LIN {X -0.130,Y -407.420,Z 765.576,A 0.000,B 0.000,C 90.000,E1 139.666} C_DIS
LIN {X -0.060,Y -413.085,Z 765.572,A 0.000,B 0.000,C 90.000,E1 138.976} C_DIS
LIN {X 0.241,Y -427.502,Z 765.564,A 0.000,B 0.000,C 90.000,E1 137.391} C_DIS
LIN {X 0.053,Y -436.215,Z 765.559,A 0.000,B 0.000,C 90.000,E1 136.539} C_DIS
LIN {X 0.009,Y -443.347,Z 765.555,A 0.000,B 0.000,C 90.000,E1 135.810} C_DIS
LIN {X -0.045,Y -451.801,Z 765.550,A 0.000,B 0.000,C 90.000,E1 134.919} C_DIS
LIN {X 0.010,Y -457.316,Z 765.546,A 0.000,B 0.000,C 90.000,E1 134.312} C_DIS
LIN {X 0.124,Y -465.443,Z 765.541,A 0.000,B 0.000,C 90.000,E1 133.380} C_DIS
LIN {X 0.124,Y -473.358,Z 765.536,A 0.000,B 0.000,C 90.000,E1 132.447} C_DIS
LIN {X -0.077,Y -480.793,Z 765.531,A 0.000,B 0.000,C 90.000,E1 131.553} C_DIS
LIN {X -0.084,Y -486.838,Z 765.527,A 0.000,B 0.000,C 90.000,E1 130.782} C_DIS
LIN {X 0.149,Y -492.370,Z 765.522,A 0.000,B 0.000,C 90.000,E1 130.011} C_DIS
LIN {X 0.158,Y -496.618,Z 765.519,A 0.000,B 0.000,C 90.000,E1 129.402} C_DIS
LIN {X 0.003,Y -502.509,Z 765.514,A 0.000,B 0.000,C 90.000,E1 128.543} C_DIS
LIN {X -0.097,Y -507.241,Z 765.510,A 0.000,B 0.000,C 90.000,E1 127.810} C_DIS
LIN {X -0.187,Y -511.626,Z 765.506,A 0.000,B 0.000,C 90.000,E1 127.076} C_DIS
LIN {X 0.175,Y -515.816,Z 765.502,A 0.000,B 0.000,C 90.000,E1 126.297} C_DIS
LIN {X -0.201,Y -521.468,Z 765.496,A 0.000,B 0.000,C 90.000,E1 125.311} C_DIS
LIN {X 0.259,Y -525.137,Z 765.492,A 0.000,B 0.000,C 90.000,E1 124.532} C_DIS
LIN {X -0.142,Y -529.163,Z 765.487,A 0.000,B 0.000,C 90.000,E1 123.706} C_DIS
LIN {X -0.224,Y -534.731,Z 765.480,A 0.000,B 0.000,C 90.000,E1 122.418} C_DIS
LIN {X -0.076,Y -538.231,Z 765.475,A 0.000,B 0.000,C 90.000,E1 121.544} C_DIS
LIN {X 0.107,Y -541.496,Z 765.471,A 0.000,B 0.000,C 90.000,E1 120.669} C_DIS
LIN {X 0.325,Y -544.507,Z 765.466,A 0.000,B 0.000,C 90.000,E1 119.795} C_DIS
LIN {X -0.175,Y -547.339,Z 765.461,A 0.000,B 0.000,C 90.000,E1 118.999} C_DIS
LIN {X 0.079,Y -550.940,Z 765.455,A 0.000,B 0.000,C 90.000,E1 117.847} C_DIS
LIN {X -0.134,Y -552.669,Z 765.452,A 0.000,B 0.000,C 90.000,E1 117.308} C_DIS
LIN {X 0.175,Y -554.965,Z 765.447,A 0.000,B 0.000,C 90.000,E1 116.437} C_DIS
LIN {X 0.048,Y -557.323,Z 765.441,A 0.000,B 0.000,C 90.000,E1 115.335} C_DIS
LIN {X 0.126,Y -558.444,Z 765.438,A 0.000,B 0.000,C 90.000,E1 114.771} C_DIS
LIN {X -0.202,Y -560.084,Z 765.432,A 0.000,B 0.000,C 90.000,E1 113.695} C_DIS
LIN {X 0.098,Y -561.976,Z 765.424,A 0.000,B 0.000,C 90.000,E1 112.280} C_DIS
LIN {X 0.121,Y -563.367,Z 765.418,A 0.000,B 0.000,C 90.000,E1 111.173} C_DIS
LIN {X -0.041,Y -564.984,Z 765.410,A 0.000,B 0.000,C 90.000,E1 109.812} C_DIS
LIN {X -0.175,Y -566.142,Z 765.404,A 0.000,B 0.000,C 90.000,E1 108.725} C_DIS
LIN {X 0.038,Y -567.477,Z 765.396,A 0.000,B 0.000,C 90.000,E1 107.330} C_DIS
LIN {X 0.267,Y -568.968,Z 765.387,A 0.000,B 0.000,C 90.000,E1 105.662} C_DIS
LIN {X -0.165,Y -570.428,Z 765.378,A 0.000,B 0.000,C 90.000,E1 104.064} C_DIS
LIN {X -0.194,Y -572.542,Z 765.366,A 0.000,B 0.000,C 90.000,E1 101.883} C_DIS
LIN {X -0.244,Y -574.082,Z 765.357,A 0.000,B 0.000,C 90.000,E1 100.254} C_DIS
LIN {X -0.098,Y -575.102,Z 765.351,A 0.000,B 0.000,C 90.000,E1 99.151} C_DIS
LIN {X 0.269,Y -576.268,Z 765.343,A 0.000,B 0.000,C 90.000,E1 97.757} C_DIS
LIN {X -0.234,Y -577.702,Z 765.333,A 0.000,B 0.000,C 90.000,E1 95.910} C_DIS
LIN {X 0.187,Y -578.800,Z 765.324,A 0.000,B 0.000,C 90.000,E1 94.245} C_DIS
LIN {X -0.104,Y -579.695,Z 765.316,A 0.000,B 0.000,C 90.000,E1 92.922} C_DIS
LIN {X -0.251,Y -580.601,Z 765.307,A 0.000,B 0.000,C 90.000,E1 91.318} C_DIS
LIN {X 0.192,Y -581.406,Z 765.298,A 0.000,B 0.000,C 90.000,E1 89.656} C_DIS
LIN {X 0.084,Y -582.021,Z 765.289,A 0.000,B 0.000,C 90.000,E1 88.051} C_DIS
LIN {X -0.182,Y -582.433,Z 765.282,A 0.000,B 0.000,C 90.000,E1 86.731} C_DIS
LIN {X -0.066,Y -582.897,Z 765.271,A 0.000,B 0.000,C 90.000,E1 84.837} C_DIS
LIN {X -0.290,Y -583.123,Z 765.264,A 0.000,B 0.000,C 90.000,E1 83.514} C_DIS
LIN {X 0.019,Y -583.259,Z 765.253,A 0.000,B 0.000,C 90.000,E1 81.602} C_DIS
LIN {X 0.060,Y -583.261,Z 765.249,A 0.000,B 0.000,C 90.000,E1 80.792} C_DIS
LIN {X -0.001,Y -583.262,Z 765.241,A 0.000,B 0.000,C 90.000,E1 79.454} C_DIS
LIN {X -0.070,Y -583.092,Z 765.234,A 0.000,B 0.000,C 90.000,E1 78.117} C_DIS
LIN {X 0.003,Y -582.582,Z 765.224,A 0.000,B 0.000,C 90.000,E1 76.228} C_DIS
LIN {X 0.178,Y -582.150,Z 765.216,A 0.000,B 0.000,C 90.000,E1 74.866} C_DIS
LIN {X -0.220,Y -581.615,Z 765.209,A 0.000,B 0.000,C 90.000,E1 73.559} C_DIS
LIN {X -0.251,Y -580.809,Z 765.200,A 0.000,B 0.000,C 90.000,E1 71.945} C_DIS
LIN {X 0.223,Y -580.086,Z 765.192,A 0.000,B 0.000,C 90.000,E1 70.550} C_DIS
LIN {X -0.250,Y -579.363,Z 765.186,A 0.000,B 0.000,C 90.000,E1 69.518} C_DIS
LIN {X -0.141,Y -578.400,Z 765.179,A 0.000,B 0.000,C 90.000,E1 68.156} C_DIS
LIN {X -0.044,Y -577.275,Z 765.171,A 0.000,B 0.000,C 90.000,E1 66.794} C_DIS
LIN {X 0.035,Y -576.497,Z 765.167,A 0.000,B 0.000,C 90.000,E1 65.973} C_DIS
LIN {X -0.286,Y -575.321,Z 765.161,A 0.000,B 0.000,C 90.000,E1 64.921} C_DIS
LIN {X -0.133,Y -574.053,Z 765.155,A 0.000,B 0.000,C 90.000,E1 63.819} C_DIS
LIN {X -0.090,Y -572.965,Z 765.150,A 0.000,B 0.000,C 90.000,E1 62.999} C_DIS
LIN {X 0.035,Y -571.306,Z 765.144,A 0.000,B 0.000,C 90.000,E1 61.897} C_DIS
LIN {X 0.135,Y -569.356,Z 765.138,A 0.000,B 0.000,C 90.000,E1 60.795} C_DIS
LIN {X -0.293,Y -567.145,Z 765.132,A 0.000,B 0.000,C 90.000,E1 59.744} C_DIS
LIN {X 0.111,Y -565.957,Z 765.129,A 0.000,B 0.000,C 90.000,E1 59.154} C_DIS
LIN {X -0.078,Y -563.214,Z 765.123,A 0.000,B 0.000,C 90.000,E1 58.074} C_DIS
LIN {X 0.002,Y -560.097,Z 765.117,A 0.000,B 0.000,C 90.000,E1 56.962} C_DIS
LIN {X -0.039,Y -557.565,Z 765.112,A 0.000,B 0.000,C 90.000,E1 56.135} C_DIS
LIN {X -0.185,Y -555.830,Z 765.109,A 0.000,B 0.000,C 90.000,E1 55.595} C_DIS
LIN {X -0.274,Y -552.875,Z 765.104,A 0.000,B 0.000,C 90.000,E1 54.769} C_DIS
LIN {X -0.076,Y -549.494,Z 765.099,A 0.000,B 0.000,C 90.000,E1 53.909} C_DIS
LIN {X -0.102,Y -546.409,Z 765.096,A 0.000,B 0.000,C 90.000,E1 53.210} C_DIS
LIN {X 0.168,Y -543.046,Z 765.092,A 0.000,B 0.000,C 90.000,E1 52.477} C_DIS
LIN {X 0.228,Y -540.213,Z 765.089,A 0.000,B 0.000,C 90.000,E1 51.904} C_DIS
LIN {X -0.155,Y -537.096,Z 765.085,A 0.000,B 0.000,C 90.000,E1 51.376} C_DIS
LIN {X 0.028,Y -532.761,Z 765.081,A 0.000,B 0.000,C 90.000,E1 50.642} C_DIS
LIN {X 0.008,Y -528.850,Z 765.078,A 0.000,B 0.000,C 90.000,E1 50.070} C_DIS
LIN {X -0.118,Y -524.929,Z 765.075,A 0.000,B 0.000,C 90.000,E1 49.542} C_DIS
LIN {X 0.141,Y -520.019,Z 765.072,A 0.000,B 0.000,C 90.000,E1 48.933} C_DIS
LIN {X -0.100,Y -516.148,Z 765.070,A 0.000,B 0.000,C 90.000,E1 48.528} C_DIS
LIN {X -0.016,Y -510.601,Z 765.066,A 0.000,B 0.000,C 90.000,E1 47.957} C_DIS
LIN {X -0.040,Y -506.284,Z 765.064,A 0.000,B 0.000,C 90.000,E1 47.553} C_DIS
LIN {X 0.083,Y -500.284,Z 765.061,A 0.000,B 0.000,C 90.000,E1 47.025} C_DIS
LIN {X 0.034,Y -495.791,Z 765.059,A 0.000,B 0.000,C 90.000,E1 46.662} C_DIS
LIN {X 0.187,Y -487.760,Z 765.056,A 0.000,B 0.000,C 90.000,E1 46.053} C_DIS
LIN {X -0.185,Y -481.381,Z 765.054,A 0.000,B 0.000,C 90.000,E1 45.648} C_DIS
LIN {X 0.041,Y -473.279,Z 765.051,A 0.000,B 0.000,C 90.000,E1 45.081} C_DIS
LIN {X 0.063,Y -463.499,Z 765.047,A 0.000,B 0.000,C 90.000,E1 44.433} C_DIS
LIN {X 0.134,Y -444.156,Z 765.040,A 0.000,B 0.000,C 90.000,E1 43.137} C_DIS
LIN {X -0.050,Y -419.026,Z 765.030,A 0.000,B 0.000,C 90.000,E1 41.353} C_DIS
LIN {X 0.070,Y -413.289,Z 765.027,A 0.000,B 0.000,C 90.000,E1 40.862} C_DIS
LIN {X -0.212,Y -409.341,Z 765.025,A 0.000,B 0.000,C 90.000,E1 40.539} C_DIS
LIN {X -0.238,Y -409.310,Z 765.025,A 0.000,B 0.000,C 90.000,E1 40.539} C_DIS
LIN {X 0.130,Y -406.118,Z 765.015,A 0.000,B 0.000,C 90.000,E1 38.624} C_DIS
LIN {X 0.096,Y -404.664,Z 765.011,A 0.000,B 0.000,C 90.000,E1 37.935} C_DIS
LIN {X 0.157,Y -399.374,Z 764.996,A 0.000,B 0.000,C 90.000,E1 35.311} C_DIS
LIN {X 0.042,Y -399.270,Z 764.994,A 0.000,B 0.000,C 90.000,E1 34.978} C_DIS
LIN {X -0.237,Y -399.849,Z 764.979,A 0.000,B 0.000,C 90.000,E1 32.212} C_DIS
LIN {X -0.249,Y -400.946,Z 764.963,A 0.000,B 0.000,C 90.000,E1 29.411} C_DIS
LIN {X 0.141,Y -402.082,Z 764.952,A 0.000,B 0.000,C 90.000,E1 27.257} C_DIS
LIN {X 0.160,Y -403.832,Z 764.936,A 0.000,B 0.000,C 90.000,E1 24.463} C_DIS
LIN {X -0.098,Y -405.866,Z 764.921,A 0.000,B 0.000,C 90.000,E1 21.716} C_DIS
LIN {X -0.097,Y -409.099,Z 764.903,A 0.000,B 0.000,C 90.000,E1 18.598} C_DIS
LIN {X -0.112,Y -412.740,Z 764.888,A 0.000,B 0.000,C 90.000,E1 15.843} C_DIS
LIN {X 0.131,Y -416.278,Z 764.875,A 0.000,B 0.000,C 90.000,E1 13.411} C_DIS
LIN {X -0.213,Y -420.108,Z 764.861,A 0.000,B 0.000,C 90.000,E1 11.074} C_DIS
LIN {X 0.219,Y -422.884,Z 764.852,A 0.000,B 0.000,C 90.000,E1 9.321} C_DIS
LIN {X 0.150,Y -425.769,Z 764.843,A 0.000,B 0.000,C 90.000,E1 7.644} C_DIS
LIN {X 0.190,Y -429.171,Z 764.831,A 0.000,B 0.000,C 90.000,E1 5.625} C_DIS
LIN {X -0.163,Y -432.714,Z 764.820,A 0.000,B 0.000,C 90.000,E1 3.669} C_DIS
LIN {X -0.145,Y -435.835,Z 764.811,A 0.000,B 0.000,C 90.000,E1 2.007} C_DIS
LIN {X -0.158,Y -440.762,Z 764.797,A 0.000,B 0.000,C 90.000,E1 359.484} C_DIS
LIN {X -0.165,Y -445.509,Z 764.784,A 0.000,B 0.000,C 90.000,E1 357.192} C_DIS
LIN {X 0.010,Y -450.602,Z 764.772,A 0.000,B 0.000,C 90.000,E1 354.894} C_DIS
LIN {X 0.002,Y -454.397,Z 764.763,A 0.000,B 0.000,C 90.000,E1 353.280} C_DIS
LIN {X -0.098,Y -457.326,Z 764.756,A 0.000,B 0.000,C 90.000,E1 352.008} C_DIS
LIN {X 0.064,Y -459.484,Z 764.750,A 0.000,B 0.000,C 90.000,E1 351.027} C_DIS
LIN {X 0.111,Y -462.231,Z 764.743,A 0.000,B 0.000,C 90.000,E1 349.746} C_DIS
LIN {X 0.002,Y -465.459,Z 764.734,A 0.000,B 0.000,C 90.000,E1 348.173} C_DIS
LIN {X 0.238,Y -470.085,Z 764.722,A 0.000,B 0.000,C 90.000,E1 345.936} C_DIS
LIN {X -0.012,Y -471.853,Z 764.719,A 0.000,B 0.000,C 90.000,E1 345.338} C_DIS
LIN {X 0.085,Y -474.238,Z 764.715,A 0.000,B 0.000,C 90.000,E1 344.700} C_DIS
LIN {X 0.057,Y -476.137,Z 764.713,A 0.000,B 0.000,C 90.000,E1 344.338} C_DIS
LIN {X 0.276,Y -479.563,Z 764.710,A 0.000,B 0.000,C 90.000,E1 343.795} C_DIS
LIN {X 0.118,Y -482.087,Z 764.708,A 0.000,B 0.000,C 90.000,E1 343.504} C_DIS
LIN {X 0.132,Y -488.837,Z 764.705,A 0.000,B 0.000,C 90.000,E1 342.851} C_DIS
LIN {X 0.042,Y -500.528,Z 764.700,A 0.000,B 0.000,C 90.000,E1 342.000} C_DIS
LIN {X 0.262,Y -520.919,Z 764.692,A 0.000,B 0.000,C 90.000,E1 340.604} C_DIS
LIN {X 0.061,Y -536.973,Z 764.687,A 0.000,B 0.000,C 90.000,E1 339.645} C_DIS
LIN {X -0.064,Y -544.553,Z 764.684,A 0.000,B 0.000,C 90.000,E1 339.156} C_DIS
LIN {X 0.005,Y -549.016,Z 764.682,A 0.000,B 0.000,C 90.000,E1 338.827} C_DIS
LIN {X 0.092,Y -554.622,Z 764.680,A 0.000,B 0.000,C 90.000,E1 338.358} C_DIS
LIN {X 0.279,Y -560.032,Z 764.677,A 0.000,B 0.000,C 90.000,E1 337.847} C_DIS
LIN {X -0.005,Y -566.398,Z 764.674,A 0.000,B 0.000,C 90.000,E1 337.230} C_DIS
LIN {X -0.127,Y -571.260,Z 764.671,A 0.000,B 0.000,C 90.000,E1 336.719} C_DIS
LIN {X -0.173,Y -575.976,Z 764.668,A 0.000,B 0.000,C 90.000,E1 336.177} C_DIS
LIN {X 0.121,Y -579.324,Z 764.665,A 0.000,B 0.000,C 90.000,E1 335.741} C_DIS
LIN {X 0.169,Y -586.780,Z 764.660,A 0.000,B 0.000,C 90.000,E1 334.793} C_DIS
LIN {X -0.119,Y -591.775,Z 764.656,A 0.000,B 0.000,C 90.000,E1 334.152} C_DIS
LIN {X 0.077,Y -598.389,Z 764.651,A 0.000,B 0.000,C 90.000,E1 333.204} C_DIS
LIN {X 0.096,Y -604.793,Z 764.646,A 0.000,B 0.000,C 90.000,E1 332.281} C_DIS
LIN {X -0.092,Y -610.829,Z 764.641,A 0.000,B 0.000,C 90.000,E1 331.385} C_DIS
LIN {X 0.059,Y -618.094,Z 764.635,A 0.000,B 0.000,C 90.000,E1 330.205} C_DIS
LIN {X 0.329,Y -622.066,Z 764.631,A 0.000,B 0.000,C 90.000,E1 329.537} C_DIS
LIN {X 0.106,Y -627.280,Z 764.626,A 0.000,B 0.000,C 90.000,E1 328.663} C_DIS
LIN {X -0.058,Y -632.249,Z 764.621,A 0.000,B 0.000,C 90.000,E1 327.788} C_DIS
LIN {X -0.184,Y -636.241,Z 764.617,A 0.000,B 0.000,C 90.000,E1 327.041} C_DIS
LIN {X 0.120,Y -641.152,Z 764.611,A 0.000,B 0.000,C 90.000,E1 326.008} C_DIS
LIN {X 0.073,Y -644.730,Z 764.607,A 0.000,B 0.000,C 90.000,E1 325.261} C_DIS
LIN {X -0.051,Y -649.086,Z 764.602,A 0.000,B 0.000,C 90.000,E1 324.276} C_DIS
LIN {X -0.120,Y -653.341,Z 764.596,A 0.000,B 0.000,C 90.000,E1 323.290} C_DIS
LIN {X -0.201,Y -656.282,Z 764.592,A 0.000,B 0.000,C 90.000,E1 322.557} C_DIS
LIN {X 0.224,Y -659.990,Z 764.586,A 0.000,B 0.000,C 90.000,E1 321.537} C_DIS
LIN {X 0.227,Y -665.115,Z 764.578,A 0.000,B 0.000,C 90.000,E1 320.070} C_DIS
LIN {X 0.251,Y -669.055,Z 764.572,A 0.000,B 0.000,C 90.000,E1 318.852} C_DIS
LIN {X -0.172,Y -672.013,Z 764.566,A 0.000,B 0.000,C 90.000,E1 317.919} C_DIS
LIN {X -0.065,Y -674.712,Z 764.561,A 0.000,B 0.000,C 90.000,E1 316.944} C_DIS
LIN {X 0.043,Y -677.208,Z 764.555,A 0.000,B 0.000,C 90.000,E1 315.972} C_DIS
LIN {X 0.190,Y -679.428,Z 764.550,A 0.000,B 0.000,C 90.000,E1 315.000} C_DIS
LIN {X 0.365,Y -681.466,Z 764.545,A 0.000,B 0.000,C 90.000,E1 314.028} C_DIS
LIN {X 0.202,Y -684.365,Z 764.537,A 0.000,B 0.000,C 90.000,E1 312.609} C_DIS
LIN {X -0.033,Y -686.068,Z 764.532,A 0.000,B 0.000,C 90.000,E1 311.676} C_DIS
LIN {X 0.327,Y -687.982,Z 764.525,A 0.000,B 0.000,C 90.000,E1 310.458} C_DIS
LIN {X -0.319,Y -689.245,Z 764.520,A 0.000,B 0.000,C 90.000,E1 309.564} C_DIS
LIN {X 0.248,Y -690.972,Z 764.512,A 0.000,B 0.000,C 90.000,E1 308.096} C_DIS
LIN {X 0.180,Y -691.967,Z 764.507,A 0.000,B 0.000,C 90.000,E1 307.156} C_DIS
LIN {X -0.237,Y -693.093,Z 764.500,A 0.000,B 0.000,C 90.000,E1 306.011} C_DIS
LIN {X 0.184,Y -694.461,Z 764.491,A 0.000,B 0.000,C 90.000,E1 304.326} C_DIS
LIN {X -0.024,Y -695.317,Z 764.484,A 0.000,B 0.000,C 90.000,E1 303.166} C_DIS
LIN {X -0.317,Y -696.581,Z 764.475,A 0.000,B 0.000,C 90.000,E1 301.544} C_DIS
LIN {X -0.151,Y -697.260,Z 764.470,A 0.000,B 0.000,C 90.000,E1 300.590} C_DIS
LIN {X -0.336,Y -697.725,Z 764.465,A 0.000,B 0.000,C 90.000,E1 299.667} C_DIS
LIN {X 0.009,Y -698.248,Z 764.457,A 0.000,B 0.000,C 90.000,E1 298.231} C_DIS
LIN {X 0.044,Y -698.857,Z 764.449,A 0.000,B 0.000,C 90.000,E1 296.821} C_DIS
LIN {X -0.270,Y -699.678,Z 764.440,A 0.000,B 0.000,C 90.000,E1 295.207} C_DIS
LIN {X -0.027,Y -699.854,Z 764.437,A 0.000,B 0.000,C 90.000,E1 294.719} C_DIS
LIN {X -0.127,Y -699.502,Z 764.435,A 0.000,B 0.000,C 90.000,E1 294.259} C_DIS
LIN {X -0.145,Y -699.209,Z 764.433,A 0.000,B 0.000,C 90.000,E1 294.027} C_DIS
LIN {X 0.385,Y -697.557,Z 764.431,A 0.000,B 0.000,C 90.000,E1 293.515} C_DIS
LIN {X -0.271,Y -696.450,Z 764.430,A 0.000,B 0.000,C 90.000,E1 293.334} C_DIS
LIN {X -0.141,Y -695.454,Z 764.429,A 0.000,B 0.000,C 90.000,E1 293.206} C_DIS
LIN {X 0.208,Y -692.700,Z 764.428,A 0.000,B 0.000,C 90.000,E1 292.950} C_DIS
LIN {X -0.126,Y -689.733,Z 764.427,A 0.000,B 0.000,C 90.000,E1 292.770} C_DIS
LIN {X 0.224,Y -688.169,Z 764.426,A 0.000,B 0.000,C 90.000,E1 292.642} C_DIS
LIN {X -0.254,Y -685.863,Z 764.425,A 0.000,B 0.000,C 90.000,E1 292.589} C_DIS
LIN {X 0.166,Y -683.099,Z 764.425,A 0.000,B 0.000,C 90.000,E1 292.461} C_DIS
LIN {X -0.088,Y -675.346,Z 764.424,A 0.000,B 0.000,C 90.000,E1 292.280} C_DIS
LIN {X -0.332,Y -665.815,Z 764.423,A 0.000,B 0.000,C 90.000,E1 292.153} C_DIS
LIN {X 0.170,Y -654.659,Z 764.422,A 0.000,B 0.000,C 90.000,E1 291.972} C_DIS
LIN {X -0.165,Y -644.827,Z 764.421,A 0.000,B 0.000,C 90.000,E1 291.844} C_DIS
LIN {X -0.058,Y -635.283,Z 764.420,A 0.000,B 0.000,C 90.000,E1 291.642} C_DIS
LIN {X 0.119,Y -610.881,Z 764.417,A 0.000,B 0.000,C 90.000,E1 291.046} C_DIS
LIN {X 0.180,Y -590.362,Z 764.414,A 0.000,B 0.000,C 90.000,E1 290.482} C_DIS
LIN {X 0.198,Y -576.156,Z 764.412,A 0.000,B 0.000,C 90.000,E1 290.066} C_DIS
LIN {X 0.235,Y -565.793,Z 764.410,A 0.000,B 0.000,C 90.000,E1 289.758} C_DIS
LIN {X 0.097,Y -559.205,Z 764.408,A 0.000,B 0.000,C 90.000,E1 289.504} C_DIS
LIN {X -0.054,Y -558.097,Z 764.408,A 0.000,B 0.000,C 90.000,E1 289.450} C_DIS
LIN {X -0.081,Y -556.387,Z 764.407,A 0.000,B 0.000,C 90.000,E1 289.268} C_DIS
LIN {X -0.246,Y -555.517,Z 764.406,A 0.000,B 0.000,C 90.000,E1 289.033} C_DIS
LIN {X 0.162,Y -555.273,Z 764.405,A 0.000,B 0.000,C 90.000,E1 288.852} C_DIS
LIN {X 0.223,Y -554.452,Z 764.395,A 0.000,B 0.000,C 90.000,E1 287.040} C_DIS
LIN {X 0.016,Y -553.541,Z 764.382,A 0.000,B 0.000,C 90.000,E1 284.828} C_DIS
LIN {X 0.212,Y -553.070,Z 764.375,A 0.000,B 0.000,C 90.000,E1 283.411} C_DIS
LIN {X -0.024,Y -552.394,Z 764.364,A 0.000,B 0.000,C 90.000,E1 281.478} C_DIS
LIN {X 0.049,Y -551.818,Z 764.354,A 0.000,B 0.000,C 90.000,E1 279.792} C_DIS
LIN {X 0.109,Y -551.212,Z 764.345,A 0.000,B 0.000,C 90.000,E1 278.106} C_DIS
LIN {X -0.037,Y -550.659,Z 764.337,A 0.000,B 0.000,C 90.000,E1 276.720} C_DIS
LIN {X 0.253,Y -550.065,Z 764.331,A 0.000,B 0.000,C 90.000,E1 275.568} C_DIS
LIN {X -0.260,Y -548.466,Z 764.317,A 0.000,B 0.000,C 90.000,E1 273.094} C_DIS
LIN {X 0.041,Y -547.498,Z 764.308,A 0.000,B 0.000,C 90.000,E1 271.375} C_DIS
LIN {X 0.225,Y -546.833,Z 764.301,A 0.000,B 0.000,C 90.000,E1 270.229} C_DIS
LIN {X -0.065,Y -545.694,Z 764.292,A 0.000,B 0.000,C 90.000,E1 268.568} C_DIS
LIN {X 0.237,Y -544.414,Z 764.281,A 0.000,B 0.000,C 90.000,E1 266.560} C_DIS
LIN {X -0.060,Y -543.363,Z 764.272,A 0.000,B 0.000,C 90.000,E1 264.894} C_DIS
LIN {X 0.120,Y -542.577,Z 764.265,A 0.000,B 0.000,C 90.000,E1 263.742} C_DIS
LIN {X -0.179,Y -541.493,Z 764.258,A 0.000,B 0.000,C 90.000,E1 262.356} C_DIS
LIN {X 0.246,Y -539.599,Z 764.245,A 0.000,B 0.000,C 90.000,E1 260.038} C_DIS
LIN {X 0.139,Y -538.181,Z 764.235,A 0.000,B 0.000,C 90.000,E1 258.342} C_DIS
LIN {X 0.002,Y -536.652,Z 764.226,A 0.000,B 0.000,C 90.000,E1 256.645} C_DIS
LIN {X 0.305,Y -535.844,Z 764.221,A 0.000,B 0.000,C 90.000,E1 255.755} C_DIS
LIN {X -0.290,Y -533.977,Z 764.212,A 0.000,B 0.000,C 90.000,E1 254.102} C_DIS
LIN {X 0.092,Y -531.401,Z 764.199,A 0.000,B 0.000,C 90.000,E1 251.764} C_DIS
LIN {X -0.016,Y -530.378,Z 764.194,A 0.000,B 0.000,C 90.000,E1 250.913} C_DIS
LIN {X -0.263,Y -527.981,Z 764.184,A 0.000,B 0.000,C 90.000,E1 249.209} C_DIS
LIN {X 0.136,Y -525.937,Z 764.176,A 0.000,B 0.000,C 90.000,E1 247.720} C_DIS
LIN {X -0.135,Y -522.848,Z 764.165,A 0.000,B 0.000,C 90.000,E1 245.717} C_DIS
LIN {X 0.058,Y -519.997,Z 764.155,A 0.000,B 0.000,C 90.000,E1 243.948} C_DIS
LIN {X -0.086,Y -518.031,Z 764.149,A 0.000,B 0.000,C 90.000,E1 242.794} C_DIS
LIN {X -0.262,Y -515.918,Z 764.142,A 0.000,B 0.000,C 90.000,E1 241.641} C_DIS
LIN {X -0.225,Y -512.513,Z 764.133,A 0.000,B 0.000,C 90.000,E1 239.871} C_DIS
LIN {X -0.112,Y -508.509,Z 764.121,A 0.000,B 0.000,C 90.000,E1 237.788} C_DIS
LIN {X -0.258,Y -506.730,Z 764.116,A 0.000,B 0.000,C 90.000,E1 236.914} C_DIS
LIN {X -0.147,Y -504.762,Z 764.111,A 0.000,B 0.000,C 90.000,E1 236.008} C_DIS
LIN {X -0.167,Y -502.008,Z 764.104,A 0.000,B 0.000,C 90.000,E1 234.815} C_DIS
LIN {X -0.107,Y -499.861,Z 764.099,A 0.000,B 0.000,C 90.000,E1 233.909} C_DIS
LIN {X -0.076,Y -497.564,Z 764.094,A 0.000,B 0.000,C 90.000,E1 233.004} C_DIS
LIN {X 0.121,Y -491.485,Z 764.081,A 0.000,B 0.000,C 90.000,E1 230.561} C_DIS
LIN {X -0.227,Y -485.840,Z 764.067,A 0.000,B 0.000,C 90.000,E1 228.162} C_DIS
LIN {X -0.039,Y -481.876,Z 764.057,A 0.000,B 0.000,C 90.000,E1 226.296} C_DIS
LIN {X 0.159,Y -477.277,Z 764.045,A 0.000,B 0.000,C 90.000,E1 224.109} C_DIS
LIN {X -0.298,Y -473.893,Z 764.037,A 0.000,B 0.000,C 90.000,E1 222.609} C_DIS
LIN {X 0.197,Y -470.468,Z 764.028,A 0.000,B 0.000,C 90.000,E1 220.987} C_DIS
LIN {X -0.115,Y -467.753,Z 764.021,A 0.000,B 0.000,C 90.000,E1 219.769} C_DIS
LIN {X -0.229,Y -463.676,Z 764.010,A 0.000,B 0.000,C 90.000,E1 217.890} C_DIS
LIN {X -0.057,Y -459.688,Z 764.000,A 0.000,B 0.000,C 90.000,E1 215.964} C_DIS
LIN {X 0.116,Y -455.160,Z 763.987,A 0.000,B 0.000,C 90.000,E1 213.706} C_DIS
LIN {X -0.059,Y -451.363,Z 763.977,A 0.000,B 0.000,C 90.000,E1 211.799} C_DIS
LIN {X -0.248,Y -448.295,Z 763.968,A 0.000,B 0.000,C 90.000,E1 210.207} C_DIS
LIN {X -0.103,Y -445.249,Z 763.959,A 0.000,B 0.000,C 90.000,E1 208.565} C_DIS
LIN {X -0.076,Y -442.843,Z 763.951,A 0.000,B 0.000,C 90.000,E1 207.257} C_DIS
LIN {X 0.009,Y -438.589,Z 763.939,A 0.000,B 0.000,C 90.000,E1 204.951} C_DIS
LIN {X -0.171,Y -433.546,Z 763.924,A 0.000,B 0.000,C 90.000,E1 202.333} C_DIS
LIN {X 0.079,Y -431.084,Z 763.917,A 0.000,B 0.000,C 90.000,E1 200.972} C_DIS
LIN {X -0.056,Y -426.654,Z 763.904,A 0.000,B 0.000,C 90.000,E1 198.652} C_DIS
LIN {X -0.146,Y -423.448,Z 763.894,A 0.000,B 0.000,C 90.000,E1 196.985} C_DIS
LIN {X -0.144,Y -417.454,Z 763.877,A 0.000,B 0.000,C 90.000,E1 193.939} C_DIS
LIN {X -0.073,Y -413.739,Z 763.866,A 0.000,B 0.000,C 90.000,E1 191.883} C_DIS
LIN {X -0.218,Y -409.552,Z 763.853,A 0.000,B 0.000,C 90.000,E1 189.500} C_DIS
LIN {X -0.119,Y -407.254,Z 763.845,A 0.000,B 0.000,C 90.000,E1 188.106} C_DIS
LIN {X -0.200,Y -402.087,Z 763.828,A 0.000,B 0.000,C 90.000,E1 184.992} C_DIS
LIN {X -0.049,Y -398.444,Z 763.814,A 0.000,B 0.000,C 90.000,E1 182.522} C_DIS
LIN {X -0.167,Y -394.375,Z 763.796,A 0.000,B 0.000,C 90.000,E1 179.370} C_DIS
LIN {X 0.118,Y -391.595,Z 763.783,A 0.000,B 0.000,C 90.000,E1 176.849} C_DIS
LIN {X 0.005,Y -389.286,Z 763.769,A 0.000,B 0.000,C 90.000,E1 174.375} C_DIS
LIN {X 0.133,Y -386.992,Z 763.751,A 0.000,B 0.000,C 90.000,E1 171.141} C_DIS
LIN {X -0.061,Y -386.296,Z 763.745,A 0.000,B 0.000,C 90.000,E1 170.095} C_DIS
LIN {X -0.026,Y -385.081,Z 763.733,A 0.000,B 0.000,C 90.000,E1 167.937} C_DIS
LIN {X 0.068,Y -383.652,Z 763.717,A 0.000,B 0.000,C 90.000,E1 165.046} C_DIS
LIN {X -0.073,Y -382.799,Z 763.705,A 0.000,B 0.000,C 90.000,E1 162.906} C_DIS
LIN {X -0.012,Y -382.166,Z 763.693,A 0.000,B 0.000,C 90.000,E1 160.732} C_DIS
LIN {X 0.097,Y -381.558,Z 763.673,A 0.000,B 0.000,C 90.000,E1 157.102} C_DIS
LIN {X 0.040,Y -381.588,Z 763.665,A 0.000,B 0.000,C 90.000,E1 155.665} C_DIS
LIN {X 0.186,Y -382.545,Z 763.641,A 0.000,B 0.000,C 90.000,E1 151.307} C_DIS
LIN {X 0.178,Y -386.494,Z 763.615,A 0.000,B 0.000,C 90.000,E1 146.628} C_DIS
LIN {X -0.052,Y -388.292,Z 763.607,A 0.000,B 0.000,C 90.000,E1 145.229} C_DIS
LIN {X 0.062,Y -390.760,Z 763.599,A 0.000,B 0.000,C 90.000,E1 143.783} C_DIS
LIN {X 0.207,Y -392.132,Z 763.595,A 0.000,B 0.000,C 90.000,E1 143.050} C_DIS
LIN {X -0.099,Y -394.909,Z 763.589,A 0.000,B 0.000,C 90.000,E1 142.029} C_DIS
LIN {X -0.071,Y -397.259,Z 763.585,A 0.000,B 0.000,C 90.000,E1 141.331} C_DIS
LIN {X 0.148,Y -399.077,Z 763.583,A 0.000,B 0.000,C 90.000,E1 140.884} C_DIS
LIN {X 0.045,Y -399.762,Z 763.582,A 0.000,B 0.000,C 90.000,E1 140.723} C_DIS
LIN {X -0.034,Y -403.659,Z 763.578,A 0.000,B 0.000,C 90.000,E1 140.033} C_DIS
LIN {X 0.042,Y -406.700,Z 763.576,A 0.000,B 0.000,C 90.000,E1 139.585} C_DIS
LIN {X -0.151,Y -413.032,Z 763.571,A 0.000,B 0.000,C 90.000,E1 138.852} C_DIS
LIN {X 0.088,Y -434.802,Z 763.559,A 0.000,B 0.000,C 90.000,E1 136.539} C_DIS
LIN {X 0.114,Y -441.938,Z 763.555,A 0.000,B 0.000,C 90.000,E1 135.810} C_DIS
LIN {X -0.049,Y -450.272,Z 763.550,A 0.000,B 0.000,C 90.000,E1 134.960} C_DIS
LIN {X 0.050,Y -455.795,Z 763.547,A 0.000,B 0.000,C 90.000,E1 134.352} C_DIS
LIN {X 0.090,Y -463.779,Z 763.542,A 0.000,B 0.000,C 90.000,E1 133.461} C_DIS
LIN {X 0.277,Y -470.241,Z 763.537,A 0.000,B 0.000,C 90.000,E1 132.690} C_DIS
LIN {X -0.097,Y -477.782,Z 763.532,A 0.000,B 0.000,C 90.000,E1 131.838} C_DIS
LIN {X 0.042,Y -483.810,Z 763.528,A 0.000,B 0.000,C 90.000,E1 131.067} C_DIS
LIN {X -0.007,Y -490.817,Z 763.523,A 0.000,B 0.000,C 90.000,E1 130.172} C_DIS
LIN {X 0.075,Y -496.186,Z 763.519,A 0.000,B 0.000,C 90.000,E1 129.402} C_DIS
LIN {X -0.048,Y -499.215,Z 763.517,A 0.000,B 0.000,C 90.000,E1 128.991} C_DIS
LIN {X -0.179,Y -504.147,Z 763.512,A 0.000,B 0.000,C 90.000,E1 128.257} C_DIS
LIN {X -0.088,Y -507.846,Z 763.509,A 0.000,B 0.000,C 90.000,E1 127.649} C_DIS
LIN {X 0.125,Y -511.406,Z 763.506,A 0.000,B 0.000,C 90.000,E1 127.030} C_DIS
LIN {X 0.075,Y -515.649,Z 763.502,A 0.000,B 0.000,C 90.000,E1 126.297} C_DIS
LIN {X -0.302,Y -521.343,Z 763.496,A 0.000,B 0.000,C 90.000,E1 125.311} C_DIS
LIN {X 0.154,Y -525.014,Z 763.492,A 0.000,B 0.000,C 90.000,E1 124.532} C_DIS
LIN {X -0.250,Y -529.091,Z 763.487,A 0.000,B 0.000,C 90.000,E1 123.706} C_DIS
LIN {X 0.256,Y -535.249,Z 763.479,A 0.000,B 0.000,C 90.000,E1 122.212} C_DIS
LIN {X -0.048,Y -538.728,Z 763.474,A 0.000,B 0.000,C 90.000,E1 121.386} C_DIS
LIN {X 0.134,Y -540.958,Z 763.471,A 0.000,B 0.000,C 90.000,E1 120.797} C_DIS
LIN {X 0.082,Y -544.961,Z 763.465,A 0.000,B 0.000,C 90.000,E1 119.667} C_DIS
LIN {X -0.179,Y -548.711,Z 763.459,A 0.000,B 0.000,C 90.000,E1 118.565} C_DIS
LIN {X -0.131,Y -552.255,Z 763.452,A 0.000,B 0.000,C 90.000,E1 117.436} C_DIS
LIN {X 0.172,Y -554.606,Z 763.448,A 0.000,B 0.000,C 90.000,E1 116.565} C_DIS
LIN {X 0.257,Y -556.509,Z 763.443,A 0.000,B 0.000,C 90.000,E1 115.720} C_DIS
LIN {X 0.118,Y -558.231,Z 763.438,A 0.000,B 0.000,C 90.000,E1 114.899} C_DIS
LIN {X -0.003,Y -559.630,Z 763.434,A 0.000,B 0.000,C 90.000,E1 114.079} C_DIS
LIN {X 0.087,Y -561.929,Z 763.425,A 0.000,B 0.000,C 90.000,E1 112.408} C_DIS
LIN {X 0.232,Y -564.000,Z 763.415,A 0.000,B 0.000,C 90.000,E1 110.737} C_DIS
LIN {X -0.116,Y -565.597,Z 763.408,A 0.000,B 0.000,C 90.000,E1 109.396} C_DIS
LIN {X -0.290,Y -567.326,Z 763.399,A 0.000,B 0.000,C 90.000,E1 107.764} C_DIS
LIN {X 0.107,Y -568.839,Z 763.389,A 0.000,B 0.000,C 90.000,E1 106.079} C_DIS
LIN {X -0.005,Y -570.615,Z 763.379,A 0.000,B 0.000,C 90.000,E1 104.175} C_DIS
LIN {X -0.156,Y -572.719,Z 763.367,A 0.000,B 0.000,C 90.000,E1 102.007} C_DIS
LIN {X -0.089,Y -574.305,Z 763.358,A 0.000,B 0.000,C 90.000,E1 100.366} C_DIS
LIN {X 0.260,Y -575.564,Z 763.350,A 0.000,B 0.000,C 90.000,E1 98.973} C_DIS
LIN {X -0.227,Y -576.533,Z 763.344,A 0.000,B 0.000,C 90.000,E1 97.936} C_DIS
LIN {X -0.280,Y -577.776,Z 763.335,A 0.000,B 0.000,C 90.000,E1 96.315} C_DIS
LIN {X -0.158,Y -578.557,Z 763.329,A 0.000,B 0.000,C 90.000,E1 95.220} C_DIS
LIN {X 0.125,Y -579.486,Z 763.321,A 0.000,B 0.000,C 90.000,E1 93.841} C_DIS
LIN {X -0.189,Y -580.375,Z 763.314,A 0.000,B 0.000,C 90.000,E1 92.522} C_DIS
LIN {X 0.260,Y -581.235,Z 763.305,A 0.000,B 0.000,C 90.000,E1 90.859} C_DIS
LIN {X -0.037,Y -581.939,Z 763.297,A 0.000,B 0.000,C 90.000,E1 89.542} C_DIS
LIN {X -0.134,Y -582.528,Z 763.289,A 0.000,B 0.000,C 90.000,E1 87.936} C_DIS
LIN {X 0.189,Y -582.947,Z 763.281,A 0.000,B 0.000,C 90.000,E1 86.560} C_DIS
LIN {X 0.145,Y -583.310,Z 763.272,A 0.000,B 0.000,C 90.000,E1 84.951} C_DIS
LIN {X -0.069,Y -583.549,Z 763.265,A 0.000,B 0.000,C 90.000,E1 83.628} C_DIS
LIN {X -0.216,Y -583.627,Z 763.257,A 0.000,B 0.000,C 90.000,E1 82.299} C_DIS
LIN {X 0.211,Y -583.731,Z 763.250,A 0.000,B 0.000,C 90.000,E1 80.914} C_DIS
LIN {X 0.148,Y -583.663,Z 763.242,A 0.000,B 0.000,C 90.000,E1 79.577} C_DIS
LIN {X 0.198,Y -583.489,Z 763.235,A 0.000,B 0.000,C 90.000,E1 78.229} C_DIS
LIN {X 0.248,Y -583.114,Z 763.227,A 0.000,B 0.000,C 90.000,E1 76.881} C_DIS
LIN {X -0.137,Y -582.738,Z 763.220,A 0.000,B 0.000,C 90.000,E1 75.574} C_DIS
LIN {X 0.041,Y -582.197,Z 763.212,A 0.000,B 0.000,C 90.000,E1 74.212} C_DIS
LIN {X -0.022,Y -581.714,Z 763.206,A 0.000,B 0.000,C 90.000,E1 73.142} C_DIS
LIN {X 0.079,Y -581.180,Z 763.200,A 0.000,B 0.000,C 90.000,E1 72.054} C_DIS
LIN {X -0.173,Y -580.432,Z 763.193,A 0.000,B 0.000,C 90.000,E1 70.732} C_DIS
LIN {X -0.250,Y -579.514,Z 763.185,A 0.000,B 0.000,C 90.000,E1 69.390} C_DIS
LIN {X -0.134,Y -578.491,Z 763.178,A 0.000,B 0.000,C 90.000,E1 68.028} C_DIS
LIN {X -0.033,Y -577.338,Z 763.170,A 0.000,B 0.000,C 90.000,E1 66.666} C_DIS
LIN {X -0.339,Y -576.238,Z 763.164,A 0.000,B 0.000,C 90.000,E1 65.613} C_DIS
LIN {X 0.035,Y -574.318,Z 763.155,A 0.000,B 0.000,C 90.000,E1 63.948} C_DIS
LIN {X 0.080,Y -573.220,Z 763.151,A 0.000,B 0.000,C 90.000,E1 63.127} C_DIS
LIN {X 0.045,Y -571.114,Z 763.143,A 0.000,B 0.000,C 90.000,E1 61.769} C_DIS
LIN {X 0.140,Y -569.070,Z 763.137,A 0.000,B 0.000,C 90.000,E1 60.667} C_DIS
LIN {X -0.006,Y -566.794,Z 763.131,A 0.000,B 0.000,C 90.000,E1 59.587} C_DIS
LIN {X 0.208,Y -564.858,Z 763.127,A 0.000,B 0.000,C 90.000,E1 58.742} C_DIS
LIN {X 0.209,Y -562.719,Z 763.122,A 0.000,B 0.000,C 90.000,E1 57.916} C_DIS
LIN {X -0.019,Y -559.470,Z 763.116,A 0.000,B 0.000,C 90.000,E1 56.834} C_DIS
LIN {X -0.152,Y -557.798,Z 763.113,A 0.000,B 0.000,C 90.000,E1 56.294} C_DIS
LIN {X -0.221,Y -555.047,Z 763.108,A 0.000,B 0.000,C 90.000,E1 55.468} C_DIS
LIN {X -0.001,Y -551.937,Z 763.103,A 0.000,B 0.000,C 90.000,E1 54.609} C_DIS
LIN {X -0.192,Y -549.716,Z 763.100,A 0.000,B 0.000,C 90.000,E1 54.069} C_DIS
LIN {X -0.035,Y -545.912,Z 763.096,A 0.000,B 0.000,C 90.000,E1 53.210} C_DIS
LIN {X 0.227,Y -542.498,Z 763.092,A 0.000,B 0.000,C 90.000,E1 52.477} C_DIS
LIN {X 0.282,Y -539.596,Z 763.089,A 0.000,B 0.000,C 90.000,E1 51.904} C_DIS
LIN {X -0.105,Y -536.409,Z 763.085,A 0.000,B 0.000,C 90.000,E1 51.376} C_DIS
LIN {X -0.094,Y -532.899,Z 763.082,A 0.000,B 0.000,C 90.000,E1 50.803} C_DIS
LIN {X 0.224,Y -528.989,Z 763.079,A 0.000,B 0.000,C 90.000,E1 50.194} C_DIS
LIN {X 0.174,Y -524.711,Z 763.076,A 0.000,B 0.000,C 90.000,E1 49.622} C_DIS
LIN {X 0.034,Y -519.861,Z 763.073,A 0.000,B 0.000,C 90.000,E1 49.057} C_DIS
LIN {X 0.050,Y -514.558,Z 763.069,A 0.000,B 0.000,C 90.000,E1 48.485} C_DIS
LIN {X 0.282,Y -510.744,Z 763.067,A 0.000,B 0.000,C 90.000,E1 48.081} C_DIS
LIN {X -0.223,Y -505.337,Z 763.065,A 0.000,B 0.000,C 90.000,E1 47.634} C_DIS
LIN {X -0.162,Y -497.662,Z 763.061,A 0.000,B 0.000,C 90.000,E1 46.986} C_DIS
LIN {X 0.162,Y -494.562,Z 763.060,A 0.000,B 0.000,C 90.000,E1 46.701} C_DIS
LIN {X 0.057,Y -486.548,Z 763.056,A 0.000,B 0.000,C 90.000,E1 46.134} C_DIS
LIN {X 0.188,Y -478.526,Z 763.053,A 0.000,B 0.000,C 90.000,E1 45.567} C_DIS
LIN {X -0.156,Y -465.577,Z 763.049,A 0.000,B 0.000,C 90.000,E1 44.757} C_DIS
LIN {X 0.044,Y -449.303,Z 763.043,A 0.000,B 0.000,C 90.000,E1 43.662} C_DIS
LIN {X 0.022,Y -423.856,Z 763.033,A 0.000,B 0.000,C 90.000,E1 41.881} C_DIS
LIN {X 0.005,Y -414.526,Z 763.029,A 0.000,B 0.000,C 90.000,E1 41.148} C_DIS
LIN {X -0.116,Y -411.557,Z 763.027,A 0.000,B 0.000,C 90.000,E1 40.906} C_DIS
LIN {X -0.099,Y -409.671,Z 763.026,A 0.000,B 0.000,C 90.000,E1 40.701} C_DIS
LIN {X -0.123,Y -409.640,Z 763.026,A 0.000,B 0.000,C 90.000,E1 40.701} C_DIS
LIN {X -0.011,Y -405.814,Z 763.014,A 0.000,B 0.000,C 90.000,E1 38.463} C_DIS
LIN {X -0.116,Y -399.683,Z 762.997,A 0.000,B 0.000,C 90.000,E1 35.518} C_DIS
LIN {X 0.104,Y -399.541,Z 762.996,A 0.000,B 0.000,C 90.000,E1 35.311} C_DIS
LIN {X 0.051,Y -400.112,Z 762.980,A 0.000,B 0.000,C 90.000,E1 32.339} C_DIS
LIN {X -0.065,Y -401.375,Z 762.962,A 0.000,B 0.000,C 90.000,E1 29.205} C_DIS
LIN {X -0.212,Y -402.503,Z 762.951,A 0.000,B 0.000,C 90.000,E1 27.129} C_DIS
LIN {X -0.116,Y -403.314,Z 762.943,A 0.000,B 0.000,C 90.000,E1 25.720} C_DIS
LIN {X -0.180,Y -404.260,Z 762.935,A 0.000,B 0.000,C 90.000,E1 24.335} C_DIS
LIN {X 0.122,Y -405.802,Z 762.924,A 0.000,B 0.000,C 90.000,E1 22.206} C_DIS
LIN {X -0.148,Y -409.257,Z 762.904,A 0.000,B 0.000,C 90.000,E1 18.779} C_DIS
LIN {X -0.024,Y -413.321,Z 762.887,A 0.000,B 0.000,C 90.000,E1 15.662} C_DIS
LIN {X 0.091,Y -416.373,Z 762.876,A 0.000,B 0.000,C 90.000,E1 13.592} C_DIS
LIN {X -0.164,Y -420.180,Z 762.862,A 0.000,B 0.000,C 90.000,E1 11.243} C_DIS
LIN {X 0.194,Y -422.949,Z 762.853,A 0.000,B 0.000,C 90.000,E1 9.500} C_DIS
LIN {X -0.199,Y -426.344,Z 762.842,A 0.000,B 0.000,C 90.000,E1 7.530} C_DIS
LIN {X -0.045,Y -430.333,Z 762.829,A 0.000,B 0.000,C 90.000,E1 5.163} C_DIS
LIN {X -0.209,Y -435.158,Z 762.814,A 0.000,B 0.000,C 90.000,E1 2.522} C_DIS
LIN {X -0.038,Y -438.913,Z 762.803,A 0.000,B 0.000,C 90.000,E1 0.516} C_DIS
LIN {X -0.040,Y -441.686,Z 762.795,A 0.000,B 0.000,C 90.000,E1 359.141} C_DIS
LIN {X 0.139,Y -447.198,Z 762.781,A 0.000,B 0.000,C 90.000,E1 356.502} C_DIS
LIN {X 0.114,Y -453.111,Z 762.766,A 0.000,B 0.000,C 90.000,E1 353.913} C_DIS
LIN {X -0.062,Y -456.117,Z 762.759,A 0.000,B 0.000,C 90.000,E1 352.648} C_DIS
LIN {X 0.090,Y -459.694,Z 762.750,A 0.000,B 0.000,C 90.000,E1 351.027} C_DIS
LIN {X 0.141,Y -462.415,Z 762.743,A 0.000,B 0.000,C 90.000,E1 349.746} C_DIS
LIN {X 0.035,Y -465.630,Z 762.734,A 0.000,B 0.000,C 90.000,E1 348.173} C_DIS
LIN {X -0.182,Y -470.097,Z 762.722,A 0.000,B 0.000,C 90.000,E1 345.992} C_DIS
LIN {X 0.026,Y -471.740,Z 762.719,A 0.000,B 0.000,C 90.000,E1 345.338} C_DIS
LIN {X -0.155,Y -472.682,Z 762.717,A 0.000,B 0.000,C 90.000,E1 345.046} C_DIS
LIN {X -0.132,Y -474.440,Z 762.714,A 0.000,B 0.000,C 90.000,E1 344.574} C_DIS
LIN {X -0.008,Y -477.199,Z 762.711,A 0.000,B 0.000,C 90.000,E1 344.031} C_DIS
LIN {X 0.041,Y -480.350,Z 762.709,A 0.000,B 0.000,C 90.000,E1 343.559} C_DIS
LIN {X -0.025,Y -483.474,Z 762.707,A 0.000,B 0.000,C 90.000,E1 343.196} C_DIS
LIN {X -0.134,Y -487.879,Z 762.704,A 0.000,B 0.000,C 90.000,E1 342.779} C_DIS
LIN {X 0.032,Y -496.029,Z 762.701,A 0.000,B 0.000,C 90.000,E1 342.127} C_DIS
LIN {X 0.100,Y -513.438,Z 762.694,A 0.000,B 0.000,C 90.000,E1 340.913} C_DIS
LIN {X 0.148,Y -527.650,Z 762.689,A 0.000,B 0.000,C 90.000,E1 340.007} C_DIS
LIN {X -0.017,Y -537.282,Z 762.686,A 0.000,B 0.000,C 90.000,E1 339.444} C_DIS
LIN {X 0.075,Y -541.908,Z 762.684,A 0.000,B 0.000,C 90.000,E1 339.135} C_DIS
LIN {X -0.003,Y -547.970,Z 762.682,A 0.000,B 0.000,C 90.000,E1 338.720} C_DIS
LIN {X -0.150,Y -553.573,Z 762.679,A 0.000,B 0.000,C 90.000,E1 338.284} C_DIS
LIN {X -0.056,Y -560.292,Z 762.676,A 0.000,B 0.000,C 90.000,E1 337.667} C_DIS
LIN {X -0.107,Y -565.433,Z 762.673,A 0.000,B 0.000,C 90.000,E1 337.155} C_DIS
LIN {X -0.025,Y -570.395,Z 762.670,A 0.000,B 0.000,C 90.000,E1 336.613} C_DIS
LIN {X 0.216,Y -575.126,Z 762.667,A 0.000,B 0.000,C 90.000,E1 336.049} C_DIS
LIN {X -0.097,Y -579.619,Z 762.664,A 0.000,B 0.000,C 90.000,E1 335.537} C_DIS
LIN {X -0.043,Y -587.054,Z 762.659,A 0.000,B 0.000,C 90.000,E1 334.588} C_DIS
LIN {X 0.205,Y -592.057,Z 762.655,A 0.000,B 0.000,C 90.000,E1 333.896} C_DIS
LIN {X -0.125,Y -598.724,Z 762.650,A 0.000,B 0.000,C 90.000,E1 332.999} C_DIS
LIN {X -0.099,Y -605.145,Z 762.645,A 0.000,B 0.000,C 90.000,E1 332.076} C_DIS
LIN {X -0.282,Y -611.201,Z 762.640,A 0.000,B 0.000,C 90.000,E1 331.179} C_DIS
LIN {X -0.135,Y -619.349,Z 762.633,A 0.000,B 0.000,C 90.000,E1 329.871} C_DIS
LIN {X 0.143,Y -624.007,Z 762.628,A 0.000,B 0.000,C 90.000,E1 329.076} C_DIS
LIN {X -0.056,Y -629.889,Z 762.623,A 0.000,B 0.000,C 90.000,E1 328.074} C_DIS
LIN {X 0.146,Y -634.704,Z 762.618,A 0.000,B 0.000,C 90.000,E1 327.168} C_DIS
LIN {X -0.060,Y -640.944,Z 762.611,A 0.000,B 0.000,C 90.000,E1 325.928} C_DIS
LIN {X -0.126,Y -644.006,Z 762.607,A 0.000,B 0.000,C 90.000,E1 325.308} C_DIS
LIN {X 0.273,Y -648.412,Z 762.602,A 0.000,B 0.000,C 90.000,E1 324.276} C_DIS
LIN {X 0.198,Y -652.750,Z 762.596,A 0.000,B 0.000,C 90.000,E1 323.290} C_DIS
LIN {X 0.113,Y -655.761,Z 762.592,A 0.000,B 0.000,C 90.000,E1 322.557} C_DIS
LIN {X -0.394,Y -659.508,Z 762.587,A 0.000,B 0.000,C 90.000,E1 321.618} C_DIS
LIN {X 0.019,Y -664.707,Z 762.578,A 0.000,B 0.000,C 90.000,E1 320.114} C_DIS
LIN {X 0.047,Y -667.945,Z 762.573,A 0.000,B 0.000,C 90.000,E1 319.138} C_DIS
LIN {X 0.113,Y -671.000,Z 762.568,A 0.000,B 0.000,C 90.000,E1 318.162} C_DIS
LIN {X -0.266,Y -674.474,Z 762.561,A 0.000,B 0.000,C 90.000,E1 316.986} C_DIS
LIN {X 0.333,Y -677.010,Z 762.556,A 0.000,B 0.000,C 90.000,E1 315.972} C_DIS
LIN {X -0.002,Y -679.281,Z 762.550,A 0.000,B 0.000,C 90.000,E1 315.040} C_DIS
LIN {X -0.310,Y -681.366,Z 762.545,A 0.000,B 0.000,C 90.000,E1 314.109} C_DIS
LIN {X -0.014,Y -684.314,Z 762.537,A 0.000,B 0.000,C 90.000,E1 312.651} C_DIS
LIN {X 0.254,Y -686.061,Z 762.532,A 0.000,B 0.000,C 90.000,E1 311.676} C_DIS
LIN {X -0.355,Y -688.019,Z 762.525,A 0.000,B 0.000,C 90.000,E1 310.539} C_DIS
LIN {X -0.030,Y -689.327,Z 762.520,A 0.000,B 0.000,C 90.000,E1 309.564} C_DIS
LIN {X -0.431,Y -691.071,Z 762.512,A 0.000,B 0.000,C 90.000,E1 308.177} C_DIS
LIN {X -0.079,Y -692.073,Z 762.507,A 0.000,B 0.000,C 90.000,E1 307.202} C_DIS
LIN {X 0.058,Y -693.219,Z 762.500,A 0.000,B 0.000,C 90.000,E1 306.011} C_DIS
LIN {X 0.090,Y -694.597,Z 762.491,A 0.000,B 0.000,C 90.000,E1 304.358} C_DIS
LIN {X 0.046,Y -695.301,Z 762.486,A 0.000,B 0.000,C 90.000,E1 303.420} C_DIS
LIN {X -0.258,Y -696.536,Z 762.477,A 0.000,B 0.000,C 90.000,E1 301.799} C_DIS
LIN {X -0.095,Y -697.237,Z 762.471,A 0.000,B 0.000,C 90.000,E1 300.846} C_DIS
LIN {X 0.321,Y -697.784,Z 762.466,A 0.000,B 0.000,C 90.000,E1 299.873} C_DIS
LIN {X 0.321,Y -698.360,Z 762.457,A 0.000,B 0.000,C 90.000,E1 298.231} C_DIS
LIN {X -0.266,Y -698.971,Z 762.449,A 0.000,B 0.000,C 90.000,E1 296.873} C_DIS
LIN {X 0.047,Y -699.780,Z 762.440,A 0.000,B 0.000,C 90.000,E1 295.207} C_DIS
LIN {X -0.345,Y -699.933,Z 762.438,A 0.000,B 0.000,C 90.000,E1 294.771} C_DIS
LIN {X 0.191,Y -699.593,Z 762.435,A 0.000,B 0.000,C 90.000,E1 294.259} C_DIS
LIN {X 0.173,Y -699.325,Z 762.434,A 0.000,B 0.000,C 90.000,E1 294.027} C_DIS
LIN {X 0.064,Y -697.660,Z 762.431,A 0.000,B 0.000,C 90.000,E1 293.567} C_DIS
LIN {X 0.047,Y -696.614,Z 762.430,A 0.000,B 0.000,C 90.000,E1 293.334} C_DIS
LIN {X 0.177,Y -695.700,Z 762.429,A 0.000,B 0.000,C 90.000,E1 293.206} C_DIS
LIN {X 0.304,Y -694.347,Z 762.428,A 0.000,B 0.000,C 90.000,E1 293.078} C_DIS
LIN {X -0.090,Y -688.331,Z 762.426,A 0.000,B 0.000,C 90.000,E1 292.695} C_DIS
LIN {X 0.027,Y -686.097,Z 762.426,A 0.000,B 0.000,C 90.000,E1 292.589} C_DIS
LIN {X -0.224,Y -683.210,Z 762.425,A 0.000,B 0.000,C 90.000,E1 292.514} C_DIS
LIN {X 0.120,Y -675.290,Z 762.424,A 0.000,B 0.000,C 90.000,E1 292.280} C_DIS
LIN {X 0.209,Y -667.803,Z 762.423,A 0.000,B 0.000,C 90.000,E1 292.153} C_DIS
LIN {X -0.177,Y -654.488,Z 762.422,A 0.000,B 0.000,C 90.000,E1 292.025} C_DIS
LIN {X 0.105,Y -644.623,Z 762.421,A 0.000,B 0.000,C 90.000,E1 291.844} C_DIS
LIN {X -0.010,Y -635.177,Z 762.420,A 0.000,B 0.000,C 90.000,E1 291.663} C_DIS
LIN {X 0.192,Y -607.389,Z 762.417,A 0.000,B 0.000,C 90.000,E1 290.972} C_DIS
LIN {X 0.361,Y -590.196,Z 762.414,A 0.000,B 0.000,C 90.000,E1 290.482} C_DIS
LIN {X -0.159,Y -575.988,Z 762.412,A 0.000,B 0.000,C 90.000,E1 290.120} C_DIS
LIN {X -0.114,Y -565.671,Z 762.410,A 0.000,B 0.000,C 90.000,E1 289.812} C_DIS
LIN {X 0.203,Y -560.412,Z 762.409,A 0.000,B 0.000,C 90.000,E1 289.577} C_DIS
LIN {X 0.291,Y -558.105,Z 762.408,A 0.000,B 0.000,C 90.000,E1 289.450} C_DIS
LIN {X -0.119,Y -556.202,Z 762.407,A 0.000,B 0.000,C 90.000,E1 289.268} C_DIS
LIN {X 0.146,Y -555.489,Z 762.406,A 0.000,B 0.000,C 90.000,E1 289.033} C_DIS
LIN {X 0.029,Y -555.240,Z 762.405,A 0.000,B 0.000,C 90.000,E1 288.906} C_DIS
LIN {X 0.085,Y -554.445,Z 762.395,A 0.000,B 0.000,C 90.000,E1 287.094} C_DIS
LIN {X 0.146,Y -553.641,Z 762.384,A 0.000,B 0.000,C 90.000,E1 285.134} C_DIS
LIN {X -0.185,Y -553.180,Z 762.376,A 0.000,B 0.000,C 90.000,E1 283.772} C_DIS
LIN {X 0.247,Y -552.497,Z 762.366,A 0.000,B 0.000,C 90.000,E1 281.771} C_DIS
LIN {X -0.222,Y -551.962,Z 762.356,A 0.000,B 0.000,C 90.000,E1 280.141} C_DIS
LIN {X -0.045,Y -551.192,Z 762.345,A 0.000,B 0.000,C 90.000,E1 278.163} C_DIS
LIN {X -0.194,Y -550.649,Z 762.338,A 0.000,B 0.000,C 90.000,E1 276.777} C_DIS
LIN {X 0.095,Y -550.055,Z 762.331,A 0.000,B 0.000,C 90.000,E1 275.625} C_DIS
LIN {X 0.129,Y -548.480,Z 762.317,A 0.000,B 0.000,C 90.000,E1 273.094} C_DIS
LIN {X -0.118,Y -547.495,Z 762.308,A 0.000,B 0.000,C 90.000,E1 271.432} C_DIS
LIN {X 0.066,Y -546.847,Z 762.302,A 0.000,B 0.000,C 90.000,E1 270.286} C_DIS
LIN {X -0.184,Y -545.525,Z 762.291,A 0.000,B 0.000,C 90.000,E1 268.339} C_DIS
LIN {X 0.141,Y -544.097,Z 762.278,A 0.000,B 0.000,C 90.000,E1 266.045} C_DIS
LIN {X -0.123,Y -543.019,Z 762.269,A 0.000,B 0.000,C 90.000,E1 264.375} C_DIS
LIN {X 0.133,Y -541.779,Z 762.259,A 0.000,B 0.000,C 90.000,E1 262.648} C_DIS
LIN {X -0.254,Y -541.058,Z 762.255,A 0.000,B 0.000,C 90.000,E1 261.837} C_DIS
LIN {X 0.245,Y -539.178,Z 762.242,A 0.000,B 0.000,C 90.000,E1 259.511} C_DIS
LIN {X -0.044,Y -537.975,Z 762.234,A 0.000,B 0.000,C 90.000,E1 258.117} C_DIS
LIN {X -0.074,Y -536.459,Z 762.224,A 0.000,B 0.000,C 90.000,E1 256.408} C_DIS
LIN {X -0.238,Y -535.308,Z 762.218,A 0.000,B 0.000,C 90.000,E1 255.283} C_DIS
LIN {X 0.286,Y -533.738,Z 762.210,A 0.000,B 0.000,C 90.000,E1 253.795} C_DIS
LIN {X -0.026,Y -531.471,Z 762.199,A 0.000,B 0.000,C 90.000,E1 251.819} C_DIS
LIN {X -0.131,Y -530.466,Z 762.194,A 0.000,B 0.000,C 90.000,E1 250.967} C_DIS
LIN {X -0.058,Y -528.516,Z 762.186,A 0.000,B 0.000,C 90.000,E1 249.518} C_DIS
LIN {X -0.163,Y -526.053,Z 762.177,A 0.000,B 0.000,C 90.000,E1 247.794} C_DIS
LIN {X 0.039,Y -522.961,Z 762.165,A 0.000,B 0.000,C 90.000,E1 245.741} C_DIS
LIN {X -0.249,Y -520.106,Z 762.156,A 0.000,B 0.000,C 90.000,E1 244.024} C_DIS
LIN {X 0.066,Y -518.136,Z 762.149,A 0.000,B 0.000,C 90.000,E1 242.820} C_DIS
LIN {X 0.127,Y -516.032,Z 762.143,A 0.000,B 0.000,C 90.000,E1 241.641} C_DIS
LIN {X 0.163,Y -512.629,Z 762.133,A 0.000,B 0.000,C 90.000,E1 239.871} C_DIS
LIN {X 0.277,Y -508.671,Z 762.121,A 0.000,B 0.000,C 90.000,E1 237.788} C_DIS
LIN {X 0.131,Y -506.851,Z 762.116,A 0.000,B 0.000,C 90.000,E1 236.914} C_DIS
LIN {X 0.136,Y -504.161,Z 762.110,A 0.000,B 0.000,C 90.000,E1 235.722} C_DIS
LIN {X -0.068,Y -502.144,Z 762.105,A 0.000,B 0.000,C 90.000,E1 234.848} C_DIS
LIN {X 0.282,Y -499.998,Z 762.100,A 0.000,B 0.000,C 90.000,E1 233.909} C_DIS
LIN {X -0.087,Y -497.722,Z 762.095,A 0.000,B 0.000,C 90.000,E1 233.050} C_DIS
LIN {X -0.183,Y -491.612,Z 762.081,A 0.000,B 0.000,C 90.000,E1 230.642} C_DIS
LIN {X 0.160,Y -485.974,Z 762.068,A 0.000,B 0.000,C 90.000,E1 228.162} C_DIS
LIN {X -0.001,Y -481.993,Z 762.057,A 0.000,B 0.000,C 90.000,E1 226.338} C_DIS
LIN {X -0.130,Y -477.411,Z 762.045,A 0.000,B 0.000,C 90.000,E1 224.190} C_DIS
LIN {X 0.088,Y -474.043,Z 762.037,A 0.000,B 0.000,C 90.000,E1 222.609} C_DIS
LIN {X -0.081,Y -470.623,Z 762.028,A 0.000,B 0.000,C 90.000,E1 221.067} C_DIS
LIN {X -0.029,Y -467.875,Z 762.021,A 0.000,B 0.000,C 90.000,E1 219.806} C_DIS
LIN {X 0.156,Y -463.805,Z 762.011,A 0.000,B 0.000,C 90.000,E1 217.890} C_DIS
LIN {X -0.044,Y -459.806,Z 762.000,A 0.000,B 0.000,C 90.000,E1 216.011} C_DIS
LIN {X -0.131,Y -455.284,Z 761.988,A 0.000,B 0.000,C 90.000,E1 213.785} C_DIS
LIN {X -0.059,Y -451.486,Z 761.977,A 0.000,B 0.000,C 90.000,E1 211.848} C_DIS
LIN {X 0.136,Y -448.424,Z 761.968,A 0.000,B 0.000,C 90.000,E1 210.207} C_DIS
LIN {X -0.109,Y -445.375,Z 761.959,A 0.000,B 0.000,C 90.000,E1 208.615} C_DIS
LIN {X -0.086,Y -442.993,Z 761.952,A 0.000,B 0.000,C 90.000,E1 207.308} C_DIS
LIN {X -0.190,Y -438.726,Z 761.939,A 0.000,B 0.000,C 90.000,E1 205.027} C_DIS
LIN {X -0.014,Y -434.323,Z 761.926,A 0.000,B 0.000,C 90.000,E1 202.695} C_DIS
LIN {X -0.092,Y -431.247,Z 761.917,A 0.000,B 0.000,C 90.000,E1 201.046} C_DIS
LIN {X -0.211,Y -426.812,Z 761.904,A 0.000,B 0.000,C 90.000,E1 198.725} C_DIS
LIN {X -0.165,Y -423.610,Z 761.895,A 0.000,B 0.000,C 90.000,E1 197.040} C_DIS
LIN {X 0.085,Y -418.247,Z 761.880,A 0.000,B 0.000,C 90.000,E1 194.300} C_DIS
LIN {X -0.177,Y -413.896,Z 761.866,A 0.000,B 0.000,C 90.000,E1 191.951} C_DIS
LIN {X 0.138,Y -410.321,Z 761.855,A 0.000,B 0.000,C 90.000,E1 189.849} C_DIS
LIN {X -0.155,Y -408.013,Z 761.847,A 0.000,B 0.000,C 90.000,E1 188.511} C_DIS
LIN {X -0.164,Y -403.364,Z 761.832,A 0.000,B 0.000,C 90.000,E1 185.739} C_DIS
LIN {X 0.022,Y -399.660,Z 761.818,A 0.000,B 0.000,C 90.000,E1 183.269} C_DIS
LIN {X -0.103,Y -394.980,Z 761.799,A 0.000,B 0.000,C 90.000,E1 179.771} C_DIS
LIN {X -0.111,Y -392.566,Z 761.787,A 0.000,B 0.000,C 90.000,E1 177.650} C_DIS
LIN {X 0.076,Y -389.765,Z 761.771,A 0.000,B 0.000,C 90.000,E1 174.780} C_DIS
LIN {X 0.155,Y -387.184,Z 761.751,A 0.000,B 0.000,C 90.000,E1 171.197} C_DIS
LIN {X -0.035,Y -386.507,Z 761.745,A 0.000,B 0.000,C 90.000,E1 170.151} C_DIS
LIN {X 0.007,Y -385.316,Z 761.733,A 0.000,B 0.000,C 90.000,E1 167.993} C_DIS
LIN {X 0.091,Y -384.261,Z 761.721,A 0.000,B 0.000,C 90.000,E1 165.825} C_DIS
LIN {X -0.028,Y -383.238,Z 761.707,A 0.000,B 0.000,C 90.000,E1 163.323} C_DIS
LIN {X 0.046,Y -382.598,Z 761.695,A 0.000,B 0.000,C 90.000,E1 161.148} C_DIS
LIN {X -0.107,Y -381.937,Z 761.677,A 0.000,B 0.000,C 90.000,E1 157.922} C_DIS
LIN {X -0.017,Y -381.886,Z 761.665,A 0.000,B 0.000,C 90.000,E1 155.741} C_DIS
LIN {X 0.129,Y -382.728,Z 761.641,A 0.000,B 0.000,C 90.000,E1 151.385} C_DIS
LIN {X 0.093,Y -385.437,Z 761.621,A 0.000,B 0.000,C 90.000,E1 147.788} C_DIS
LIN {X -0.114,Y -388.219,Z 761.607,A 0.000,B 0.000,C 90.000,E1 145.308} C_DIS
LIN {X 0.216,Y -392.606,Z 761.593,A 0.000,B 0.000,C 90.000,E1 142.763} C_DIS
LIN {X -0.172,Y -394.442,Z 761.589,A 0.000,B 0.000,C 90.000,E1 142.110} C_DIS
LIN {X 0.007,Y -396.611,Z 761.585,A 0.000,B 0.000,C 90.000,E1 141.376} C_DIS
LIN {X -0.045,Y -399.341,Z 761.582,A 0.000,B 0.000,C 90.000,E1 140.678} C_DIS
LIN {X -0.131,Y -403.120,Z 761.578,A 0.000,B 0.000,C 90.000,E1 139.989} C_DIS
LIN {X -0.186,Y -406.137,Z 761.575,A 0.000,B 0.000,C 90.000,E1 139.542} C_DIS
LIN {X -0.142,Y -411.750,Z 761.571,A 0.000,B 0.000,C 90.000,E1 138.852} C_DIS
LIN {X 0.058,Y -435.075,Z 761.558,A 0.000,B 0.000,C 90.000,E1 136.377} C_DIS
LIN {X -0.051,Y -440.856,Z 761.555,A 0.000,B 0.000,C 90.000,E1 135.810} C_DIS
LIN {X 0.169,Y -449.217,Z 761.550,A 0.000,B 0.000,C 90.000,E1 134.919} C_DIS
LIN {X 0.233,Y -457.420,Z 761.545,A 0.000,B 0.000,C 90.000,E1 134.028} C_DIS
LIN {X -0.009,Y -463.962,Z 761.541,A 0.000,B 0.000,C 90.000,E1 133.338} C_DIS
LIN {X -0.005,Y -469.285,Z 761.537,A 0.000,B 0.000,C 90.000,E1 132.732} C_DIS
LIN {X 0.020,Y -476.875,Z 761.532,A 0.000,B 0.000,C 90.000,E1 131.838} C_DIS
LIN {X 0.185,Y -481.760,Z 761.529,A 0.000,B 0.000,C 90.000,E1 131.229} C_DIS
LIN {X 0.013,Y -490.226,Z 761.523,A 0.000,B 0.000,C 90.000,E1 130.172} C_DIS
LIN {X -0.057,Y -497.914,Z 761.517,A 0.000,B 0.000,C 90.000,E1 129.116} C_DIS
LIN {X -0.203,Y -503.045,Z 761.513,A 0.000,B 0.000,C 90.000,E1 128.382} C_DIS
LIN {X 0.175,Y -508.601,Z 761.508,A 0.000,B 0.000,C 90.000,E1 127.443} C_DIS
LIN {X 0.099,Y -513.040,Z 761.504,A 0.000,B 0.000,C 90.000,E1 126.710} C_DIS
LIN {X 0.108,Y -518.876,Z 761.498,A 0.000,B 0.000,C 90.000,E1 125.678} C_DIS
LIN {X -0.005,Y -522.044,Z 761.495,A 0.000,B 0.000,C 90.000,E1 125.105} C_DIS
LIN {X -0.270,Y -525.619,Z 761.491,A 0.000,B 0.000,C 90.000,E1 124.405} C_DIS
LIN {X 0.095,Y -528.450,Z 761.488,A 0.000,B 0.000,C 90.000,E1 123.785} C_DIS
LIN {X 0.144,Y -534.667,Z 761.480,A 0.000,B 0.000,C 90.000,E1 122.339} C_DIS
LIN {X 0.292,Y -538.182,Z 761.475,A 0.000,B 0.000,C 90.000,E1 121.465} C_DIS
LIN {X 0.007,Y -540.458,Z 761.472,A 0.000,B 0.000,C 90.000,E1 120.924} C_DIS
LIN {X -0.053,Y -544.509,Z 761.466,A 0.000,B 0.000,C 90.000,E1 119.795} C_DIS
LIN {X -0.075,Y -547.384,Z 761.461,A 0.000,B 0.000,C 90.000,E1 118.949} C_DIS
LIN {X -0.302,Y -551.003,Z 761.455,A 0.000,B 0.000,C 90.000,E1 117.847} C_DIS
LIN {X -0.024,Y -552.743,Z 761.451,A 0.000,B 0.000,C 90.000,E1 117.257} C_DIS
LIN {X 0.040,Y -555.058,Z 761.447,A 0.000,B 0.000,C 90.000,E1 116.411} C_DIS
LIN {X 0.169,Y -557.473,Z 761.441,A 0.000,B 0.000,C 90.000,E1 115.283} C_DIS
LIN {X -0.256,Y -558.587,Z 761.438,A 0.000,B 0.000,C 90.000,E1 114.771} C_DIS
LIN {X 0.137,Y -559.947,Z 761.433,A 0.000,B 0.000,C 90.000,E1 113.898} C_DIS
LIN {X 0.139,Y -561.911,Z 761.425,A 0.000,B 0.000,C 90.000,E1 112.514} C_DIS
LIN {X 0.070,Y -564.000,Z 761.416,A 0.000,B 0.000,C 90.000,E1 110.865} C_DIS
LIN {X 0.120,Y -565.340,Z 761.410,A 0.000,B 0.000,C 90.000,E1 109.758} C_DIS
LIN {X -0.212,Y -566.833,Z 761.402,A 0.000,B 0.000,C 90.000,E1 108.417} C_DIS
LIN {X -0.160,Y -568.203,Z 761.395,A 0.000,B 0.000,C 90.000,E1 107.040} C_DIS
LIN {X 0.093,Y -569.747,Z 761.385,A 0.000,B 0.000,C 90.000,E1 105.371} C_DIS
LIN {X 0.048,Y -571.051,Z 761.378,A 0.000,B 0.000,C 90.000,E1 104.008} C_DIS
LIN {X 0.044,Y -573.191,Z 761.366,A 0.000,B 0.000,C 90.000,E1 101.827} C_DIS
LIN {X 0.011,Y -574.806,Z 761.357,A 0.000,B 0.000,C 90.000,E1 100.197} C_DIS
LIN {X -0.191,Y -576.071,Z 761.349,A 0.000,B 0.000,C 90.000,E1 98.859} C_DIS
LIN {X 0.112,Y -577.241,Z 761.342,A 0.000,B 0.000,C 90.000,E1 97.473} C_DIS
LIN {X 0.219,Y -578.731,Z 761.331,A 0.000,B 0.000,C 90.000,E1 95.568} C_DIS
LIN {X 0.135,Y -579.826,Z 761.322,A 0.000,B 0.000,C 90.000,E1 93.955} C_DIS
LIN {X -0.176,Y -580.746,Z 761.315,A 0.000,B 0.000,C 90.000,E1 92.636} C_DIS
LIN {X -0.127,Y -581.810,Z 761.304,A 0.000,B 0.000,C 90.000,E1 90.745} C_DIS
LIN {X -0.239,Y -582.569,Z 761.295,A 0.000,B 0.000,C 90.000,E1 89.141} C_DIS
LIN {X 0.258,Y -583.126,Z 761.286,A 0.000,B 0.000,C 90.000,E1 87.478} C_DIS
LIN {X 0.002,Y -583.516,Z 761.279,A 0.000,B 0.000,C 90.000,E1 86.159} C_DIS
LIN {X 0.016,Y -583.854,Z 761.270,A 0.000,B 0.000,C 90.000,E1 84.546} C_DIS
LIN {X -0.187,Y -584.035,Z 761.262,A 0.000,B 0.000,C 90.000,E1 83.223} C_DIS
LIN {X 0.064,Y -584.166,Z 761.252,A 0.000,B 0.000,C 90.000,E1 81.319} C_DIS
LIN {X 0.010,Y -584.096,Z 761.244,A 0.000,B 0.000,C 90.000,E1 79.982} C_DIS
LIN {X 0.069,Y -583.940,Z 761.237,A 0.000,B 0.000,C 90.000,E1 78.634} C_DIS
LIN {X -0.232,Y -583.715,Z 761.231,A 0.000,B 0.000,C 90.000,E1 77.589} C_DIS
LIN {X -0.142,Y -583.139,Z 761.221,A 0.000,B 0.000,C 90.000,E1 75.700} C_DIS
LIN {X 0.038,Y -582.573,Z 761.213,A 0.000,B 0.000,C 90.000,E1 74.338} C_DIS
LIN {X -0.024,Y -582.103,Z 761.207,A 0.000,B 0.000,C 90.000,E1 73.268} C_DIS
LIN {X -0.264,Y -581.388,Z 761.200,A 0.000,B 0.000,C 90.000,E1 71.945} C_DIS
LIN {X 0.220,Y -580.601,Z 761.192,A 0.000,B 0.000,C 90.000,E1 70.550} C_DIS
LIN {X 0.144,Y -579.657,Z 761.185,A 0.000,B 0.000,C 90.000,E1 69.209} C_DIS
LIN {X -0.128,Y -578.809,Z 761.179,A 0.000,B 0.000,C 90.000,E1 68.156} C_DIS
LIN {X -0.024,Y -577.629,Z 761.171,A 0.000,B 0.000,C 90.000,E1 66.794} C_DIS
LIN {X 0.059,Y -576.806,Z 761.167,A 0.000,B 0.000,C 90.000,E1 65.973} C_DIS
LIN {X -0.258,Y -575.571,Z 761.161,A 0.000,B 0.000,C 90.000,E1 64.921} C_DIS
LIN {X -0.102,Y -574.235,Z 761.155,A 0.000,B 0.000,C 90.000,E1 63.819} C_DIS
LIN {X -0.057,Y -573.047,Z 761.150,A 0.000,B 0.000,C 90.000,E1 62.999} C_DIS
LIN {X 0.069,Y -571.340,Z 761.144,A 0.000,B 0.000,C 90.000,E1 61.897} C_DIS
LIN {X 0.341,Y -569.870,Z 761.139,A 0.000,B 0.000,C 90.000,E1 61.051} C_DIS
LIN {X -0.079,Y -567.584,Z 761.133,A 0.000,B 0.000,C 90.000,E1 59.999} C_DIS
LIN {X 0.143,Y -565.719,Z 761.129,A 0.000,B 0.000,C 90.000,E1 59.154} C_DIS
LIN {X -0.049,Y -562.890,Z 761.123,A 0.000,B 0.000,C 90.000,E1 58.074} C_DIS
LIN {X 0.025,Y -559.639,Z 761.117,A 0.000,B 0.000,C 90.000,E1 56.962} C_DIS
LIN {X -0.021,Y -557.032,Z 761.112,A 0.000,B 0.000,C 90.000,E1 56.135} C_DIS
LIN {X -0.170,Y -555.204,Z 761.109,A 0.000,B 0.000,C 90.000,E1 55.595} C_DIS
LIN {X -0.265,Y -552.076,Z 761.104,A 0.000,B 0.000,C 90.000,E1 54.769} C_DIS
LIN {X -0.136,Y -549.814,Z 761.101,A 0.000,B 0.000,C 90.000,E1 54.196} C_DIS
LIN {X -0.113,Y -545.341,Z 761.096,A 0.000,B 0.000,C 90.000,E1 53.210} C_DIS
LIN {X 0.145,Y -541.873,Z 761.092,A 0.000,B 0.000,C 90.000,E1 52.477} C_DIS
LIN {X 0.020,Y -539.716,Z 761.089,A 0.000,B 0.000,C 90.000,E1 52.065} C_DIS
LIN {X -0.194,Y -535.595,Z 761.085,A 0.000,B 0.000,C 90.000,E1 51.376} C_DIS
LIN {X -0.189,Y -531.995,Z 761.082,A 0.000,B 0.000,C 90.000,E1 50.803} C_DIS
LIN {X 0.124,Y -528.003,Z 761.079,A 0.000,B 0.000,C 90.000,E1 50.194} C_DIS
LIN {X 0.066,Y -523.527,Z 761.076,A 0.000,B 0.000,C 90.000,E1 49.622} C_DIS
LIN {X -0.080,Y -518.532,Z 761.073,A 0.000,B 0.000,C 90.000,E1 49.057} C_DIS
LIN {X -0.091,Y -514.692,Z 761.070,A 0.000,B 0.000,C 90.000,E1 48.647} C_DIS
LIN {X 0.092,Y -508.098,Z 761.067,A 0.000,B 0.000,C 90.000,E1 48.000} C_DIS
LIN {X -0.185,Y -503.670,Z 761.065,A 0.000,B 0.000,C 90.000,E1 47.634} C_DIS
LIN {X 0.037,Y -497.612,Z 761.062,A 0.000,B 0.000,C 90.000,E1 47.106} C_DIS
LIN {X 0.013,Y -492.832,Z 761.060,A 0.000,B 0.000,C 90.000,E1 46.743} C_DIS
LIN {X 0.017,Y -484.881,Z 761.057,A 0.000,B 0.000,C 90.000,E1 46.176} C_DIS
LIN {X -0.134,Y -476.758,Z 761.054,A 0.000,B 0.000,C 90.000,E1 45.648} C_DIS
LIN {X 0.192,Y -463.699,Z 761.049,A 0.000,B 0.000,C 90.000,E1 44.757} C_DIS
LIN {X 0.269,Y -449.114,Z 761.044,A 0.000,B 0.000,C 90.000,E1 43.785} C_DIS
LIN {X 0.226,Y -433.103,Z 761.037,A 0.000,B 0.000,C 90.000,E1 42.690} C_DIS
LIN {X -0.094,Y -418.707,Z 761.031,A 0.000,B 0.000,C 90.000,E1 41.676} C_DIS
LIN {X 0.165,Y -412.778,Z 761.029,A 0.000,B 0.000,C 90.000,E1 41.148} C_DIS
LIN {X 0.053,Y -410.098,Z 761.027,A 0.000,B 0.000,C 90.000,E1 40.906} C_DIS
LIN {X 0.026,Y -410.066,Z 761.027,A 0.000,B 0.000,C 90.000,E1 40.906} C_DIS
LIN {X -0.025,Y -406.084,Z 761.015,A 0.000,B 0.000,C 90.000,E1 38.624} C_DIS
LIN {X 0.078,Y -403.856,Z 761.009,A 0.000,B 0.000,C 90.000,E1 37.569} C_DIS
LIN {X -0.112,Y -399.983,Z 760.998,A 0.000,B 0.000,C 90.000,E1 35.678} C_DIS
LIN {X -0.216,Y -399.839,Z 760.997,A 0.000,B 0.000,C 90.000,E1 35.518} C_DIS
LIN {X 0.079,Y -400.378,Z 760.981,A 0.000,B 0.000,C 90.000,E1 32.498} C_DIS
LIN {X -0.055,Y -401.483,Z 760.965,A 0.000,B 0.000,C 90.000,E1 29.716} C_DIS
LIN {X 0.044,Y -402.747,Z 760.952,A 0.000,B 0.000,C 90.000,E1 27.257} C_DIS
LIN {X -0.142,Y -403.761,Z 760.942,A 0.000,B 0.000,C 90.000,E1 25.540} C_DIS
LIN {X -0.030,Y -404.689,Z 760.934,A 0.000,B 0.000,C 90.000,E1 24.131} C_DIS
LIN {X 0.212,Y -407.265,Z 760.917,A 0.000,B 0.000,C 90.000,E1 20.972} C_DIS
LIN {X 0.020,Y -409.043,Z 760.907,A 0.000,B 0.000,C 90.000,E1 19.268} C_DIS
LIN {X 0.145,Y -412.965,Z 760.890,A 0.000,B 0.000,C 90.000,E1 16.150} C_DIS
LIN {X 0.148,Y -416.998,Z 760.875,A 0.000,B 0.000,C 90.000,E1 13.411} C_DIS
LIN {X 0.169,Y -420.268,Z 760.863,A 0.000,B 0.000,C 90.000,E1 11.366} C_DIS
LIN {X -0.147,Y -423.556,Z 760.852,A 0.000,B 0.000,C 90.000,E1 9.378} C_DIS
LIN {X -0.207,Y -426.365,Z 760.843,A 0.000,B 0.000,C 90.000,E1 7.701} C_DIS
LIN {X -0.157,Y -429.765,Z 760.831,A 0.000,B 0.000,C 90.000,E1 5.682} C_DIS
LIN {X 0.121,Y -434.533,Z 760.817,A 0.000,B 0.000,C 90.000,E1 2.980} C_DIS
LIN {X -0.163,Y -438.241,Z 760.806,A 0.000,B 0.000,C 90.000,E1 1.031} C_DIS
LIN {X -0.038,Y -441.949,Z 760.795,A 0.000,B 0.000,C 90.000,E1 359.141} C_DIS
LIN {X 0.150,Y -447.460,Z 760.781,A 0.000,B 0.000,C 90.000,E1 356.502} C_DIS
LIN {X 0.132,Y -453.331,Z 760.766,A 0.000,B 0.000,C 90.000,E1 353.913} C_DIS
LIN {X 0.179,Y -457.056,Z 760.757,A 0.000,B 0.000,C 90.000,E1 352.299} C_DIS
LIN {X 0.117,Y -459.894,Z 760.750,A 0.000,B 0.000,C 90.000,E1 351.027} C_DIS
LIN {X 0.170,Y -462.613,Z 760.743,A 0.000,B 0.000,C 90.000,E1 349.746} C_DIS
LIN {X 0.068,Y -465.808,Z 760.734,A 0.000,B 0.000,C 90.000,E1 348.173} C_DIS
LIN {X -0.070,Y -469.493,Z 760.724,A 0.000,B 0.000,C 90.000,E1 346.297} C_DIS
LIN {X 0.064,Y -471.615,Z 760.719,A 0.000,B 0.000,C 90.000,E1 345.338} C_DIS
LIN {X 0.160,Y -473.546,Z 760.715,A 0.000,B 0.000,C 90.000,E1 344.700} C_DIS
LIN {X -0.142,Y -475.374,Z 760.713,A 0.000,B 0.000,C 90.000,E1 344.267} C_DIS
LIN {X 0.144,Y -476.924,Z 760.711,A 0.000,B 0.000,C 90.000,E1 343.921} C_DIS
LIN {X 0.257,Y -480.284,Z 760.708,A 0.000,B 0.000,C 90.000,E1 343.378} C_DIS
LIN {X 0.099,Y -482.790,Z 760.706,A 0.000,B 0.000,C 90.000,E1 343.087} C_DIS
LIN {X -0.142,Y -489.046,Z 760.703,A 0.000,B 0.000,C 90.000,E1 342.489} C_DIS
LIN {X 0.039,Y -500.769,Z 760.698,A 0.000,B 0.000,C 90.000,E1 341.583} C_DIS
LIN {X -0.233,Y -521.238,Z 760.690,A 0.000,B 0.000,C 90.000,E1 340.242} C_DIS
LIN {X -0.116,Y -537.195,Z 760.685,A 0.000,B 0.000,C 90.000,E1 339.263} C_DIS
LIN {X 0.049,Y -541.676,Z 760.683,A 0.000,B 0.000,C 90.000,E1 338.954} C_DIS
LIN {X 0.004,Y -546.294,Z 760.681,A 0.000,B 0.000,C 90.000,E1 338.646} C_DIS
LIN {X -0.162,Y -550.554,Z 760.680,A 0.000,B 0.000,C 90.000,E1 338.337} C_DIS
LIN {X -0.115,Y -556.218,Z 760.677,A 0.000,B 0.000,C 90.000,E1 337.847} C_DIS
LIN {X 0.222,Y -561.209,Z 760.674,A 0.000,B 0.000,C 90.000,E1 337.358} C_DIS
LIN {X -0.103,Y -566.358,Z 760.672,A 0.000,B 0.000,C 90.000,E1 336.869} C_DIS
LIN {X 0.043,Y -572.495,Z 760.668,A 0.000,B 0.000,C 90.000,E1 336.177} C_DIS
LIN {X 0.112,Y -579.396,Z 760.663,A 0.000,B 0.000,C 90.000,E1 335.357} C_DIS
LIN {X 0.226,Y -585.776,Z 760.659,A 0.000,B 0.000,C 90.000,E1 334.537} C_DIS
LIN {X -0.070,Y -590.867,Z 760.655,A 0.000,B 0.000,C 90.000,E1 333.896} C_DIS
LIN {X 0.117,Y -597.679,Z 760.650,A 0.000,B 0.000,C 90.000,E1 332.948} C_DIS
LIN {X 0.127,Y -604.176,Z 760.645,A 0.000,B 0.000,C 90.000,E1 332.025} C_DIS
LIN {X -0.069,Y -610.306,Z 760.640,A 0.000,B 0.000,C 90.000,E1 331.129} C_DIS
LIN {X 0.070,Y -617.758,Z 760.633,A 0.000,B 0.000,C 90.000,E1 329.950} C_DIS
LIN {X -0.203,Y -622.526,Z 760.629,A 0.000,B 0.000,C 90.000,E1 329.203} C_DIS
LIN {X -0.087,Y -629.239,Z 760.622,A 0.000,B 0.000,C 90.000,E1 328.043} C_DIS
LIN {X 0.295,Y -633.493,Z 760.618,A 0.000,B 0.000,C 90.000,E1 327.248} C_DIS
LIN {X 0.083,Y -640.466,Z 760.611,A 0.000,B 0.000,C 90.000,E1 325.881} C_DIS
LIN {X 0.030,Y -644.154,Z 760.606,A 0.000,B 0.000,C 90.000,E1 325.135} C_DIS
LIN {X 0.236,Y -650.816,Z 760.598,A 0.000,B 0.000,C 90.000,E1 323.623} C_DIS
LIN {X 0.192,Y -654.963,Z 760.593,A 0.000,B 0.000,C 90.000,E1 322.637} C_DIS
LIN {X 0.082,Y -658.794,Z 760.587,A 0.000,B 0.000,C 90.000,E1 321.662} C_DIS
LIN {X 0.125,Y -662.305,Z 760.582,A 0.000,B 0.000,C 90.000,E1 320.678} C_DIS
LIN {X 0.114,Y -665.765,Z 760.576,A 0.000,B 0.000,C 90.000,E1 319.703} C_DIS
LIN {X -0.357,Y -668.930,Z 760.571,A 0.000,B 0.000,C 90.000,E1 318.771} C_DIS
LIN {X 0.154,Y -671.224,Z 760.567,A 0.000,B 0.000,C 90.000,E1 318.000} C_DIS
LIN {X -0.219,Y -674.693,Z 760.560,A 0.000,B 0.000,C 90.000,E1 316.824} C_DIS
LIN {X 0.383,Y -677.257,Z 760.555,A 0.000,B 0.000,C 90.000,E1 315.810} C_DIS
LIN {X -0.387,Y -680.057,Z 760.548,A 0.000,B 0.000,C 90.000,E1 314.676} C_DIS
LIN {X -0.254,Y -681.613,Z 760.544,A 0.000,B 0.000,C 90.000,E1 313.947} C_DIS
LIN {X -0.418,Y -684.607,Z 760.536,A 0.000,B 0.000,C 90.000,E1 312.528} C_DIS
LIN {X -0.139,Y -686.348,Z 760.531,A 0.000,B 0.000,C 90.000,E1 311.553} C_DIS
LIN {X -0.290,Y -688.308,Z 760.524,A 0.000,B 0.000,C 90.000,E1 310.378} C_DIS
LIN {X 0.036,Y -689.617,Z 760.519,A 0.000,B 0.000,C 90.000,E1 309.402} C_DIS
LIN {X 0.180,Y -691.350,Z 760.511,A 0.000,B 0.000,C 90.000,E1 307.971} C_DIS
LIN {X 0.121,Y -692.357,Z 760.506,A 0.000,B 0.000,C 90.000,E1 307.030} C_DIS
LIN {X 0.071,Y -693.302,Z 760.501,A 0.000,B 0.000,C 90.000,E1 306.091} C_DIS
LIN {X -0.069,Y -694.671,Z 760.491,A 0.000,B 0.000,C 90.000,E1 304.452} C_DIS
LIN {X -0.279,Y -695.552,Z 760.485,A 0.000,B 0.000,C 90.000,E1 303.293} C_DIS
LIN {X -0.226,Y -696.621,Z 760.477,A 0.000,B 0.000,C 90.000,E1 301.878} C_DIS
LIN {X -0.058,Y -697.339,Z 760.472,A 0.000,B 0.000,C 90.000,E1 300.924} C_DIS
LIN {X -0.241,Y -697.896,Z 760.467,A 0.000,B 0.000,C 90.000,E1 300.001} C_DIS
LIN {X 0.109,Y -698.384,Z 760.459,A 0.000,B 0.000,C 90.000,E1 298.565} C_DIS
LIN {X 0.113,Y -699.049,Z 760.450,A 0.000,B 0.000,C 90.000,E1 296.924} C_DIS
LIN {X 0.120,Y -699.870,Z 760.441,A 0.000,B 0.000,C 90.000,E1 295.283} C_DIS
LIN {X 0.025,Y -699.999,Z 760.438,A 0.000,B 0.000,C 90.000,E1 294.823} C_DIS
LIN {X 0.001,Y -699.946,Z 760.437,A 0.000,B 0.000,C 90.000,E1 294.591} C_DIS
LIN {X -0.098,Y -699.484,Z 760.434,A 0.000,B 0.000,C 90.000,E1 294.131} C_DIS
LIN {X -0.117,Y -698.859,Z 760.433,A 0.000,B 0.000,C 90.000,E1 293.898} C_DIS
LIN {X 0.150,Y -697.992,Z 760.431,A 0.000,B 0.000,C 90.000,E1 293.643} C_DIS
LIN {X 0.412,Y -696.905,Z 760.430,A 0.000,B 0.000,C 90.000,E1 293.387} C_DIS
LIN {X -0.375,Y -696.206,Z 760.430,A 0.000,B 0.000,C 90.000,E1 293.334} C_DIS
LIN {X -0.245,Y -695.164,Z 760.429,A 0.000,B 0.000,C 90.000,E1 293.206} C_DIS
LIN {X 0.371,Y -690.539,Z 760.427,A 0.000,B 0.000,C 90.000,E1 292.823} C_DIS
LIN {X 0.225,Y -687.415,Z 760.426,A 0.000,B 0.000,C 90.000,E1 292.642} C_DIS
LIN {X -0.281,Y -684.827,Z 760.425,A 0.000,B 0.000,C 90.000,E1 292.589} C_DIS
LIN {X -0.235,Y -680.388,Z 760.425,A 0.000,B 0.000,C 90.000,E1 292.461} C_DIS
LIN {X -0.326,Y -675.106,Z 760.424,A 0.000,B 0.000,C 90.000,E1 292.333} C_DIS
LIN {X 0.245,Y -666.414,Z 760.423,A 0.000,B 0.000,C 90.000,E1 292.153} C_DIS
LIN {X -0.186,Y -656.695,Z 760.423,A 0.000,B 0.000,C 90.000,E1 292.078} C_DIS
LIN {X 0.200,Y -646.623,Z 760.422,A 0.000,B 0.000,C 90.000,E1 291.897} C_DIS
LIN {X 0.144,Y -637.132,Z 760.421,A 0.000,B 0.000,C 90.000,E1 291.716} C_DIS
LIN {X 0.212,Y -616.618,Z 760.418,A 0.000,B 0.000,C 90.000,E1 291.227} C_DIS
LIN {X 0.163,Y -595.817,Z 760.415,A 0.000,B 0.000,C 90.000,E1 290.684} C_DIS
LIN {X 0.200,Y -578.401,Z 760.412,A 0.000,B 0.000,C 90.000,E1 290.174} C_DIS
LIN {X 0.083,Y -567.890,Z 760.411,A 0.000,B 0.000,C 90.000,E1 289.885} C_DIS
LIN {X 0.084,Y -562.137,Z 760.409,A 0.000,B 0.000,C 90.000,E1 289.685} C_DIS
LIN {X -0.039,Y -559.386,Z 760.409,A 0.000,B 0.000,C 90.000,E1 289.577} C_DIS
LIN {X -0.003,Y -558.057,Z 760.408,A 0.000,B 0.000,C 90.000,E1 289.504} C_DIS
LIN {X 0.051,Y -556.046,Z 760.407,A 0.000,B 0.000,C 90.000,E1 289.268} C_DIS
LIN {X -0.209,Y -555.350,Z 760.406,A 0.000,B 0.000,C 90.000,E1 289.087} C_DIS
LIN {X -0.066,Y -554.936,Z 760.403,A 0.000,B 0.000,C 90.000,E1 288.489} C_DIS
LIN {X 0.194,Y -554.532,Z 760.397,A 0.000,B 0.000,C 90.000,E1 287.347} C_DIS
LIN {X -0.116,Y -553.736,Z 760.386,A 0.000,B 0.000,C 90.000,E1 285.426} C_DIS
LIN {X 0.209,Y -553.144,Z 760.376,A 0.000,B 0.000,C 90.000,E1 283.716} C_DIS
LIN {X 0.104,Y -552.492,Z 760.365,A 0.000,B 0.000,C 90.000,E1 281.771} C_DIS
LIN {X 0.178,Y -551.925,Z 760.356,A 0.000,B 0.000,C 90.000,E1 280.084} C_DIS
LIN {X 0.244,Y -551.256,Z 760.347,A 0.000,B 0.000,C 90.000,E1 278.398} C_DIS
LIN {X 0.209,Y -550.610,Z 760.338,A 0.000,B 0.000,C 90.000,E1 276.720} C_DIS
LIN {X -0.050,Y -550.017,Z 760.331,A 0.000,B 0.000,C 90.000,E1 275.625} C_DIS
LIN {X -0.141,Y -548.765,Z 760.320,A 0.000,B 0.000,C 90.000,E1 273.669} C_DIS
LIN {X 0.173,Y -547.813,Z 760.311,A 0.000,B 0.000,C 90.000,E1 271.949} C_DIS
LIN {X -0.080,Y -546.842,Z 760.302,A 0.000,B 0.000,C 90.000,E1 270.286} C_DIS
LIN {X 0.216,Y -545.511,Z 760.291,A 0.000,B 0.000,C 90.000,E1 268.282} C_DIS
LIN {X -0.034,Y -544.253,Z 760.280,A 0.000,B 0.000,C 90.000,E1 266.331} C_DIS
LIN {X 0.202,Y -543.219,Z 760.270,A 0.000,B 0.000,C 90.000,E1 264.609} C_DIS
LIN {X -0.017,Y -541.992,Z 760.261,A 0.000,B 0.000,C 90.000,E1 262.932} C_DIS
LIN {X 0.136,Y -541.043,Z 760.254,A 0.000,B 0.000,C 90.000,E1 261.781} C_DIS
LIN {X -0.044,Y -539.623,Z 760.245,A 0.000,B 0.000,C 90.000,E1 260.095} C_DIS
LIN {X 0.206,Y -538.474,Z 760.237,A 0.000,B 0.000,C 90.000,E1 258.645} C_DIS
LIN {X 0.184,Y -536.965,Z 760.228,A 0.000,B 0.000,C 90.000,E1 256.937} C_DIS
LIN {X -0.103,Y -535.938,Z 760.221,A 0.000,B 0.000,C 90.000,E1 255.825} C_DIS
LIN {X -0.046,Y -534.052,Z 760.212,A 0.000,B 0.000,C 90.000,E1 254.102} C_DIS
LIN {X -0.167,Y -531.484,Z 760.199,A 0.000,B 0.000,C 90.000,E1 251.819} C_DIS
LIN {X 0.229,Y -530.473,Z 760.194,A 0.000,B 0.000,C 90.000,E1 250.913} C_DIS
LIN {X -0.198,Y -528.522,Z 760.186,A 0.000,B 0.000,C 90.000,E1 249.518} C_DIS
LIN {X -0.302,Y -526.086,Z 760.177,A 0.000,B 0.000,C 90.000,E1 247.794} C_DIS
LIN {X -0.099,Y -522.996,Z 760.165,A 0.000,B 0.000,C 90.000,E1 245.741} C_DIS
LIN {X 0.083,Y -520.132,Z 760.156,A 0.000,B 0.000,C 90.000,E1 243.973} C_DIS
LIN {X -0.069,Y -518.140,Z 760.149,A 0.000,B 0.000,C 90.000,E1 242.820} C_DIS
LIN {X -0.008,Y -516.017,Z 760.143,A 0.000,B 0.000,C 90.000,E1 241.641} C_DIS
LIN {X 0.029,Y -512.630,Z 760.133,A 0.000,B 0.000,C 90.000,E1 239.871} C_DIS
LIN {X 0.144,Y -508.666,Z 760.121,A 0.000,B 0.000,C 90.000,E1 237.788} C_DIS
LIN {X -0.002,Y -506.824,Z 760.116,A 0.000,B 0.000,C 90.000,E1 236.914} C_DIS
LIN {X 0.109,Y -504.888,Z 760.111,A 0.000,B 0.000,C 90.000,E1 236.008} C_DIS
LIN {X -0.024,Y -501.423,Z 760.103,A 0.000,B 0.000,C 90.000,E1 234.529} C_DIS
LIN {X 0.030,Y -499.211,Z 760.098,A 0.000,B 0.000,C 90.000,E1 233.623} C_DIS
LIN {X -0.082,Y -496.140,Z 760.091,A 0.000,B 0.000,C 90.000,E1 232.431} C_DIS
LIN {X 0.072,Y -490.161,Z 760.078,A 0.000,B 0.000,C 90.000,E1 229.989} C_DIS
LIN {X 0.178,Y -485.279,Z 760.066,A 0.000,B 0.000,C 90.000,E1 227.838} C_DIS
LIN {X 0.220,Y -481.959,Z 760.057,A 0.000,B 0.000,C 90.000,E1 226.296} C_DIS
LIN {X -0.039,Y -478.037,Z 760.047,A 0.000,B 0.000,C 90.000,E1 224.474} C_DIS
LIN {X -0.141,Y -474.732,Z 760.038,A 0.000,B 0.000,C 90.000,E1 222.933} C_DIS
LIN {X 0.021,Y -471.331,Z 760.030,A 0.000,B 0.000,C 90.000,E1 221.353} C_DIS
LIN {X -0.086,Y -467.183,Z 760.019,A 0.000,B 0.000,C 90.000,E1 219.483} C_DIS
LIN {X 0.034,Y -463.785,Z 760.011,A 0.000,B 0.000,C 90.000,E1 217.890} C_DIS
LIN {X -0.165,Y -459.801,Z 760.000,A 0.000,B 0.000,C 90.000,E1 216.011} C_DIS
LIN {X 0.021,Y -455.939,Z 759.989,A 0.000,B 0.000,C 90.000,E1 214.072} C_DIS
LIN {X 0.114,Y -452.122,Z 759.979,A 0.000,B 0.000,C 90.000,E1 212.133} C_DIS
LIN {X 0.019,Y -448.449,Z 759.968,A 0.000,B 0.000,C 90.000,E1 210.207} C_DIS
LIN {X 0.229,Y -444.800,Z 759.957,A 0.000,B 0.000,C 90.000,E1 208.231} C_DIS
LIN {X 0.043,Y -442.384,Z 759.950,A 0.000,B 0.000,C 90.000,E1 206.950} C_DIS
LIN {X 0.095,Y -438.706,Z 759.939,A 0.000,B 0.000,C 90.000,E1 204.975} C_DIS
LIN {X -0.126,Y -434.346,Z 759.926,A 0.000,B 0.000,C 90.000,E1 202.695} C_DIS
LIN {X -0.203,Y -431.266,Z 759.917,A 0.000,B 0.000,C 90.000,E1 201.046} C_DIS
LIN {X 0.084,Y -426.832,Z 759.904,A 0.000,B 0.000,C 90.000,E1 198.671} C_DIS
LIN {X 0.132,Y -423.623,Z 759.895,A 0.000,B 0.000,C 90.000,E1 196.985} C_DIS
LIN {X -0.076,Y -418.914,Z 759.881,A 0.000,B 0.000,C 90.000,E1 194.647} C_DIS
LIN {X 0.078,Y -414.549,Z 759.868,A 0.000,B 0.000,C 90.000,E1 192.243} C_DIS
LIN {X 0.037,Y -410.409,Z 759.855,A 0.000,B 0.000,C 90.000,E1 189.849} C_DIS
LIN {X 0.170,Y -407.474,Z 759.845,A 0.000,B 0.000,C 90.000,E1 188.106} C_DIS
LIN {X 0.137,Y -402.901,Z 759.830,A 0.000,B 0.000,C 90.000,E1 185.334} C_DIS
LIN {X -0.149,Y -398.747,Z 759.814,A 0.000,B 0.000,C 90.000,E1 182.579} C_DIS
LIN {X 0.074,Y -394.276,Z 759.795,A 0.000,B 0.000,C 90.000,E1 179.026} C_DIS
LIN {X 0.120,Y -392.294,Z 759.785,A 0.000,B 0.000,C 90.000,E1 177.249} C_DIS
LIN {X -0.004,Y -389.864,Z 759.771,A 0.000,B 0.000,C 90.000,E1 174.780} C_DIS
LIN {X 0.018,Y -387.126,Z 759.749,A 0.000,B 0.000,C 90.000,E1 170.849} C_DIS
LIN {X 0.004,Y -385.909,Z 759.737,A 0.000,B 0.000,C 90.000,E1 168.701} C_DIS
LIN {X 0.099,Y -384.881,Z 759.725,A 0.000,B 0.000,C 90.000,E1 166.533} C_DIS
LIN {X -0.003,Y -383.781,Z 759.711,A 0.000,B 0.000,C 90.000,E1 164.031} C_DIS
LIN {X -0.013,Y -382.984,Z 759.697,A 0.000,B 0.000,C 90.000,E1 161.511} C_DIS
LIN {X -0.142,Y -382.276,Z 759.677,A 0.000,B 0.000,C 90.000,E1 157.922} C_DIS
LIN {X 0.109,Y -382.170,Z 759.663,A 0.000,B 0.000,C 90.000,E1 155.357} C_DIS
LIN {X -0.065,Y -383.167,Z 759.639,A 0.000,B 0.000,C 90.000,E1 151.051} C_DIS
LIN {X 0.089,Y -385.614,Z 759.621,A 0.000,B 0.000,C 90.000,E1 147.788} C_DIS
LIN {X -0.114,Y -388.296,Z 759.607,A 0.000,B 0.000,C 90.000,E1 145.308} C_DIS
LIN {X 0.217,Y -392.524,Z 759.593,A 0.000,B 0.000,C 90.000,E1 142.763} C_DIS
LIN {X -0.086,Y -395.250,Z 759.587,A 0.000,B 0.000,C 90.000,E1 141.743} C_DIS
LIN {X 0.108,Y -397.487,Z 759.583,A 0.000,B 0.000,C 90.000,E1 141.009} C_DIS
LIN {X -0.060,Y -399.460,Z 759.581,A 0.000,B 0.000,C 90.000,E1 140.517} C_DIS
LIN {X -0.144,Y -403.245,Z 759.577,A 0.000,B 0.000,C 90.000,E1 139.828} C_DIS
LIN {X -0.020,Y -405.472,Z 759.575,A 0.000,B 0.000,C 90.000,E1 139.461} C_DIS
LIN {X 0.168,Y -410.091,Z 759.572,A 0.000,B 0.000,C 90.000,E1 138.852} C_DIS
LIN {X 0.013,Y -417.279,Z 759.567,A 0.000,B 0.000,C 90.000,E1 138.081} C_DIS
LIN {X -0.191,Y -434.834,Z 759.557,A 0.000,B 0.000,C 90.000,E1 136.296} C_DIS
LIN {X -0.100,Y -442.036,Z 759.553,A 0.000,B 0.000,C 90.000,E1 135.567} C_DIS
LIN {X 0.064,Y -450.453,Z 759.548,A 0.000,B 0.000,C 90.000,E1 134.676} C_DIS
LIN {X 0.026,Y -458.846,Z 759.543,A 0.000,B 0.000,C 90.000,E1 133.785} C_DIS
LIN {X -0.290,Y -468.348,Z 759.537,A 0.000,B 0.000,C 90.000,E1 132.771} C_DIS
LIN {X -0.148,Y -477.580,Z 759.531,A 0.000,B 0.000,C 90.000,E1 131.676} C_DIS
LIN {X -0.220,Y -482.674,Z 759.528,A 0.000,B 0.000,C 90.000,E1 131.067} C_DIS
LIN {X 0.232,Y -490.019,Z 759.523,A 0.000,B 0.000,C 90.000,E1 130.092} C_DIS
LIN {X 0.160,Y -497.814,Z 759.517,A 0.000,B 0.000,C 90.000,E1 129.036} C_DIS
LIN {X 0.121,Y -502.907,Z 759.513,A 0.000,B 0.000,C 90.000,E1 128.302} C_DIS
LIN {X 0.047,Y -507.582,Z 759.509,A 0.000,B 0.000,C 90.000,E1 127.569} C_DIS
LIN {X -0.150,Y -511.232,Z 759.505,A 0.000,B 0.000,C 90.000,E1 126.996} C_DIS
LIN {X 0.093,Y -514.734,Z 759.502,A 0.000,B 0.000,C 90.000,E1 126.377} C_DIS
LIN {X -0.172,Y -521.329,Z 759.496,A 0.000,B 0.000,C 90.000,E1 125.231} C_DIS
LIN {X -0.114,Y -527.017,Z 759.489,A 0.000,B 0.000,C 90.000,E1 124.072} C_DIS
LIN {X -0.018,Y -529.021,Z 759.487,A 0.000,B 0.000,C 90.000,E1 123.627} C_DIS
LIN {X -0.104,Y -534.663,Z 759.480,A 0.000,B 0.000,C 90.000,E1 122.339} C_DIS
LIN {X 0.037,Y -539.319,Z 759.473,A 0.000,B 0.000,C 90.000,E1 121.180} C_DIS
LIN {X -0.243,Y -540.484,Z 759.472,A 0.000,B 0.000,C 90.000,E1 120.924} C_DIS
LIN {X 0.167,Y -544.550,Z 759.465,A 0.000,B 0.000,C 90.000,E1 119.745} C_DIS
LIN {X -0.329,Y -547.431,Z 759.461,A 0.000,B 0.000,C 90.000,E1 118.949} C_DIS
LIN {X 0.189,Y -551.088,Z 759.454,A 0.000,B 0.000,C 90.000,E1 117.769} C_DIS
LIN {X -0.278,Y -552.815,Z 759.451,A 0.000,B 0.000,C 90.000,E1 117.257} C_DIS
LIN {X 0.283,Y -555.119,Z 759.447,A 0.000,B 0.000,C 90.000,E1 116.360} C_DIS
LIN {X 0.129,Y -557.020,Z 759.442,A 0.000,B 0.000,C 90.000,E1 115.540} C_DIS
LIN {X -0.002,Y -558.685,Z 759.437,A 0.000,B 0.000,C 90.000,E1 114.719} C_DIS
LIN {X -0.118,Y -560.064,Z 759.433,A 0.000,B 0.000,C 90.000,E1 113.898} C_DIS
LIN {X -0.114,Y -562.053,Z 759.425,A 0.000,B 0.000,C 90.000,E1 112.514} C_DIS
LIN {X 0.225,Y -563.832,Z 759.417,A 0.000,B 0.000,C 90.000,E1 111.099} C_DIS
LIN {X -0.129,Y -565.537,Z 759.410,A 0.000,B 0.000,C 90.000,E1 109.758} C_DIS
LIN {X 0.080,Y -567.057,Z 759.402,A 0.000,B 0.000,C 90.000,E1 108.362} C_DIS
LIN {X 0.141,Y -568.443,Z 759.394,A 0.000,B 0.000,C 90.000,E1 106.985} C_DIS
LIN {X 0.228,Y -569.751,Z 759.387,A 0.000,B 0.000,C 90.000,E1 105.607} C_DIS
LIN {X 0.182,Y -571.114,Z 759.379,A 0.000,B 0.000,C 90.000,E1 104.245} C_DIS
LIN {X 0.182,Y -573.243,Z 759.367,A 0.000,B 0.000,C 90.000,E1 102.063} C_DIS
LIN {X 0.154,Y -574.910,Z 759.358,A 0.000,B 0.000,C 90.000,E1 100.433} C_DIS
LIN {X 0.167,Y -576.469,Z 759.349,A 0.000,B 0.000,C 90.000,E1 98.803} C_DIS
LIN {X 0.116,Y -577.837,Z 759.340,A 0.000,B 0.000,C 90.000,E1 97.182} C_DIS
LIN {X 0.023,Y -579.146,Z 759.331,A 0.000,B 0.000,C 90.000,E1 95.568} C_DIS
LIN {X -0.255,Y -580.091,Z 759.323,A 0.000,B 0.000,C 90.000,E1 94.245} C_DIS
LIN {X 0.056,Y -581.016,Z 759.316,A 0.000,B 0.000,C 90.000,E1 92.865} C_DIS
LIN {X -0.063,Y -581.920,Z 759.307,A 0.000,B 0.000,C 90.000,E1 91.260} C_DIS
LIN {X -0.122,Y -582.397,Z 759.303,A 0.000,B 0.000,C 90.000,E1 90.458} C_DIS
LIN {X 0.183,Y -583.052,Z 759.295,A 0.000,B 0.000,C 90.000,E1 89.083} C_DIS
LIN {X 0.107,Y -583.591,Z 759.286,A 0.000,B 0.000,C 90.000,E1 87.478} C_DIS
LIN {X -0.141,Y -584.006,Z 759.279,A 0.000,B 0.000,C 90.000,E1 86.159} C_DIS
LIN {X 0.053,Y -584.356,Z 759.268,A 0.000,B 0.000,C 90.000,E1 84.261} C_DIS
LIN {X -0.078,Y -584.509,Z 759.261,A 0.000,B 0.000,C 90.000,E1 82.932} C_DIS
LIN {X 0.189,Y -584.639,Z 759.250,A 0.000,B 0.000,C 90.000,E1 81.027} C_DIS
LIN {X 0.146,Y -584.495,Z 759.243,A 0.000,B 0.000,C 90.000,E1 79.690} C_DIS
LIN {X -0.116,Y -584.218,Z 759.234,A 0.000,B 0.000,C 90.000,E1 78.105} C_DIS
LIN {X 0.284,Y -583.910,Z 759.228,A 0.000,B 0.000,C 90.000,E1 76.992} C_DIS
LIN {X -0.227,Y -583.503,Z 759.220,A 0.000,B 0.000,C 90.000,E1 75.700} C_DIS
LIN {X 0.186,Y -582.788,Z 759.212,A 0.000,B 0.000,C 90.000,E1 74.047} C_DIS
LIN {X -0.097,Y -582.427,Z 759.207,A 0.000,B 0.000,C 90.000,E1 73.268} C_DIS
LIN {X 0.061,Y -581.526,Z 759.198,A 0.000,B 0.000,C 90.000,E1 71.638} C_DIS
LIN {X 0.004,Y -580.687,Z 759.191,A 0.000,B 0.000,C 90.000,E1 70.296} C_DIS
LIN {X 0.115,Y -579.479,Z 759.182,A 0.000,B 0.000,C 90.000,E1 68.666} C_DIS
LIN {X -0.312,Y -578.287,Z 759.174,A 0.000,B 0.000,C 90.000,E1 67.358} C_DIS
LIN {X 0.157,Y -577.279,Z 759.168,A 0.000,B 0.000,C 90.000,E1 66.230} C_DIS
LIN {X -0.061,Y -575.701,Z 759.161,A 0.000,B 0.000,C 90.000,E1 64.897} C_DIS
LIN {X -0.148,Y -574.303,Z 759.155,A 0.000,B 0.000,C 90.000,E1 63.819} C_DIS
LIN {X -0.262,Y -572.676,Z 759.148,A 0.000,B 0.000,C 90.000,E1 62.743} C_DIS
LIN {X -0.141,Y -570.837,Z 759.142,A 0.000,B 0.000,C 90.000,E1 61.641} C_DIS
LIN {X 0.124,Y -569.269,Z 759.138,A 0.000,B 0.000,C 90.000,E1 60.795} C_DIS
LIN {X -0.305,Y -566.868,Z 759.132,A 0.000,B 0.000,C 90.000,E1 59.744} C_DIS
LIN {X 0.198,Y -564.886,Z 759.127,A 0.000,B 0.000,C 90.000,E1 58.869} C_DIS
LIN {X -0.097,Y -562.691,Z 759.123,A 0.000,B 0.000,C 90.000,E1 58.074} C_DIS
LIN {X -0.116,Y -560.258,Z 759.118,A 0.000,B 0.000,C 90.000,E1 57.248} C_DIS
LIN {X -0.156,Y -557.662,Z 759.113,A 0.000,B 0.000,C 90.000,E1 56.421} C_DIS
LIN {X -0.225,Y -554.832,Z 759.109,A 0.000,B 0.000,C 90.000,E1 55.595} C_DIS
LIN {X -0.006,Y -551.627,Z 759.104,A 0.000,B 0.000,C 90.000,E1 54.736} C_DIS
LIN {X -0.007,Y -548.709,Z 759.100,A 0.000,B 0.000,C 90.000,E1 54.036} C_DIS
LIN {X -0.040,Y -545.437,Z 759.096,A 0.000,B 0.000,C 90.000,E1 53.336} C_DIS
LIN {X -0.109,Y -541.923,Z 759.092,A 0.000,B 0.000,C 90.000,E1 52.637} C_DIS
LIN {X -0.058,Y -538.982,Z 759.089,A 0.000,B 0.000,C 90.000,E1 52.065} C_DIS
LIN {X 0.303,Y -535.674,Z 759.086,A 0.000,B 0.000,C 90.000,E1 51.457} C_DIS
LIN {X -0.278,Y -531.032,Z 759.082,A 0.000,B 0.000,C 90.000,E1 50.803} C_DIS
LIN {X 0.029,Y -526.936,Z 759.079,A 0.000,B 0.000,C 90.000,E1 50.194} C_DIS
LIN {X -0.035,Y -522.296,Z 759.076,A 0.000,B 0.000,C 90.000,E1 49.622} C_DIS
LIN {X 0.060,Y -518.603,Z 759.073,A 0.000,B 0.000,C 90.000,E1 49.175} C_DIS
LIN {X 0.074,Y -513.121,Z 759.070,A 0.000,B 0.000,C 90.000,E1 48.609} C_DIS
LIN {X -0.250,Y -508.874,Z 759.068,A 0.000,B 0.000,C 90.000,E1 48.243} C_DIS
LIN {X -0.209,Y -502.889,Z 759.065,A 0.000,B 0.000,C 90.000,E1 47.715} C_DIS
LIN {X 0.053,Y -496.758,Z 759.062,A 0.000,B 0.000,C 90.000,E1 47.187} C_DIS
LIN {X 0.125,Y -492.068,Z 759.060,A 0.000,B 0.000,C 90.000,E1 46.824} C_DIS
LIN {X -0.206,Y -483.985,Z 759.057,A 0.000,B 0.000,C 90.000,E1 46.296} C_DIS
LIN {X 0.034,Y -475.884,Z 759.054,A 0.000,B 0.000,C 90.000,E1 45.729} C_DIS
LIN {X 0.016,Y -459.701,Z 759.048,A 0.000,B 0.000,C 90.000,E1 44.676} C_DIS
LIN {X -0.035,Y -441.857,Z 759.042,A 0.000,B 0.000,C 90.000,E1 43.500} C_DIS
LIN {X -0.006,Y -435.356,Z 759.039,A 0.000,B 0.000,C 90.000,E1 43.056} C_DIS
LIN {X -0.203,Y -427.718,Z 759.036,A 0.000,B 0.000,C 90.000,E1 42.528} C_DIS
LIN {X -0.283,Y -418.200,Z 759.032,A 0.000,B 0.000,C 90.000,E1 41.838} C_DIS
LIN {X -0.099,Y -413.676,Z 759.030,A 0.000,B 0.000,C 90.000,E1 41.434} C_DIS
LIN {X -0.202,Y -410.486,Z 759.029,A 0.000,B 0.000,C 90.000,E1 41.148} C_DIS
LIN {X -0.234,Y -410.462,Z 759.028,A 0.000,B 0.000,C 90.000,E1 41.148} C_DIS
LIN {X 0.246,Y -405.885,Z 759.014,A 0.000,B 0.000,C 90.000,E1 38.463} C_DIS
LIN {X -0.081,Y -400.141,Z 758.998,A 0.000,B 0.000,C 90.000,E1 35.724} C_DIS
LIN {X 0.106,Y -400.997,Z 758.976,A 0.000,B 0.000,C 90.000,E1 31.671} C_DIS
LIN {X 0.238,Y -402.062,Z 758.962,A 0.000,B 0.000,C 90.000,E1 29.205} C_DIS
LIN {X 0.071,Y -403.599,Z 758.947,A 0.000,B 0.000,C 90.000,E1 26.437} C_DIS
LIN {X -0.135,Y -405.641,Z 758.930,A 0.000,B 0.000,C 90.000,E1 23.334} C_DIS
LIN {X 0.047,Y -407.419,Z 758.918,A 0.000,B 0.000,C 90.000,E1 21.227} C_DIS
LIN {X 0.120,Y -409.550,Z 758.906,A 0.000,B 0.000,C 90.000,E1 19.141} C_DIS
LIN {X 0.121,Y -412.991,Z 758.891,A 0.000,B 0.000,C 90.000,E1 16.386} C_DIS
LIN {X 0.124,Y -416.993,Z 758.876,A 0.000,B 0.000,C 90.000,E1 13.647} C_DIS
LIN {X 0.080,Y -419.707,Z 758.867,A 0.000,B 0.000,C 90.000,E1 11.951} C_DIS
LIN {X -0.167,Y -423.550,Z 758.853,A 0.000,B 0.000,C 90.000,E1 9.613} C_DIS
LIN {X -0.037,Y -427.411,Z 758.840,A 0.000,B 0.000,C 90.000,E1 7.239} C_DIS
LIN {X 0.037,Y -430.793,Z 758.829,A 0.000,B 0.000,C 90.000,E1 5.220} C_DIS
LIN {X -0.113,Y -435.598,Z 758.814,A 0.000,B 0.000,C 90.000,E1 2.579} C_DIS
LIN {X 0.179,Y -440.021,Z 758.801,A 0.000,B 0.000,C 90.000,E1 0.229} C_DIS
LIN {X 0.172,Y -445.611,Z 758.786,A 0.000,B 0.000,C 90.000,E1 357.478} C_DIS
LIN {X 0.028,Y -449.134,Z 758.777,A 0.000,B 0.000,C 90.000,E1 355.869} C_DIS
LIN {X 0.151,Y -453.530,Z 758.766,A 0.000,B 0.000,C 90.000,E1 353.913} C_DIS
LIN {X 0.202,Y -457.277,Z 758.757,A 0.000,B 0.000,C 90.000,E1 352.299} C_DIS
LIN {X 0.143,Y -460.092,Z 758.750,A 0.000,B 0.000,C 90.000,E1 351.027} C_DIS
LIN {X 0.199,Y -462.812,Z 758.743,A 0.000,B 0.000,C 90.000,E1 349.746} C_DIS
LIN {X 0.101,Y -465.986,Z 758.734,A 0.000,B 0.000,C 90.000,E1 348.173} C_DIS
LIN {X -0.113,Y -468.423,Z 758.727,A 0.000,B 0.000,C 90.000,E1 346.937} C_DIS
LIN {X 0.167,Y -470.874,Z 758.720,A 0.000,B 0.000,C 90.000,E1 345.644} C_DIS
LIN {X -0.077,Y -472.408,Z 758.717,A 0.000,B 0.000,C 90.000,E1 345.046} C_DIS
LIN {X 0.148,Y -474.422,Z 758.713,A 0.000,B 0.000,C 90.000,E1 344.393} C_DIS
LIN {X -0.027,Y -475.588,Z 758.712,A 0.000,B 0.000,C 90.000,E1 344.102} C_DIS
LIN {X 0.145,Y -477.870,Z 758.709,A 0.000,B 0.000,C 90.000,E1 343.614} C_DIS
LIN {X -0.181,Y -481.298,Z 758.706,A 0.000,B 0.000,C 90.000,E1 343.142} C_DIS
LIN {X 0.266,Y -483.828,Z 758.705,A 0.000,B 0.000,C 90.000,E1 342.779} C_DIS
LIN {X -0.181,Y -489.001,Z 758.702,A 0.000,B 0.000,C 90.000,E1 342.308} C_DIS
LIN {X 0.193,Y -496.994,Z 758.698,A 0.000,B 0.000,C 90.000,E1 341.638} C_DIS
LIN {X -0.150,Y -514.106,Z 758.692,A 0.000,B 0.000,C 90.000,E1 340.496} C_DIS
LIN {X -0.267,Y -526.958,Z 758.687,A 0.000,B 0.000,C 90.000,E1 339.699} C_DIS
LIN {X -0.014,Y -539.783,Z 758.683,A 0.000,B 0.000,C 90.000,E1 338.901} C_DIS
LIN {X 0.033,Y -544.317,Z 758.681,A 0.000,B 0.000,C 90.000,E1 338.592} C_DIS
LIN {X 0.056,Y -550.147,Z 758.679,A 0.000,B 0.000,C 90.000,E1 338.156} C_DIS
LIN {X -0.202,Y -555.733,Z 758.676,A 0.000,B 0.000,C 90.000,E1 337.720} C_DIS
LIN {X -0.182,Y -562.299,Z 758.673,A 0.000,B 0.000,C 90.000,E1 337.102} C_DIS
LIN {X 0.220,Y -567.364,Z 758.670,A 0.000,B 0.000,C 90.000,E1 336.538} C_DIS
LIN {X -0.297,Y -572.216,Z 758.667,A 0.000,B 0.000,C 90.000,E1 336.049} C_DIS
LIN {X -0.262,Y -579.222,Z 758.662,A 0.000,B 0.000,C 90.000,E1 335.229} C_DIS
LIN {X -0.218,Y -586.681,Z 758.657,A 0.000,B 0.000,C 90.000,E1 334.280} C_DIS
LIN {X -0.135,Y -594.672,Z 758.651,A 0.000,B 0.000,C 90.000,E1 333.204} C_DIS
LIN {X -0.163,Y -601.385,Z 758.646,A 0.000,B 0.000,C 90.000,E1 332.281} C_DIS
LIN {X -0.363,Y -606.817,Z 758.642,A 0.000,B 0.000,C 90.000,E1 331.513} C_DIS
LIN {X -0.239,Y -612.838,Z 758.637,A 0.000,B 0.000,C 90.000,E1 330.589} C_DIS
LIN {X -0.049,Y -619.437,Z 758.631,A 0.000,B 0.000,C 90.000,E1 329.537} C_DIS
LIN {X 0.231,Y -624.110,Z 758.627,A 0.000,B 0.000,C 90.000,E1 328.742} C_DIS
LIN {X 0.033,Y -630.087,Z 758.621,A 0.000,B 0.000,C 90.000,E1 327.740} C_DIS
LIN {X -0.127,Y -633.526,Z 758.617,A 0.000,B 0.000,C 90.000,E1 327.120} C_DIS
LIN {X -0.361,Y -639.977,Z 758.610,A 0.000,B 0.000,C 90.000,E1 325.881} C_DIS
LIN {X -0.075,Y -643.078,Z 758.607,A 0.000,B 0.000,C 90.000,E1 325.229} C_DIS
LIN {X 0.268,Y -649.897,Z 758.599,A 0.000,B 0.000,C 90.000,E1 323.703} C_DIS
LIN {X 0.156,Y -653.105,Z 758.594,A 0.000,B 0.000,C 90.000,E1 322.970} C_DIS
LIN {X 0.087,Y -658.062,Z 758.588,A 0.000,B 0.000,C 90.000,E1 321.743} C_DIS
LIN {X 0.060,Y -663.456,Z 758.579,A 0.000,B 0.000,C 90.000,E1 320.275} C_DIS
LIN {X 0.069,Y -666.805,Z 758.574,A 0.000,B 0.000,C 90.000,E1 319.299} C_DIS
LIN {X 0.123,Y -670.702,Z 758.567,A 0.000,B 0.000,C 90.000,E1 318.081} C_DIS
LIN {X -0.259,Y -674.267,Z 758.560,A 0.000,B 0.000,C 90.000,E1 316.905} C_DIS
LIN {X 0.336,Y -676.897,Z 758.555,A 0.000,B 0.000,C 90.000,E1 315.891} C_DIS
LIN {X 0.000,Y -679.204,Z 758.550,A 0.000,B 0.000,C 90.000,E1 314.960} C_DIS
LIN {X -0.354,Y -680.866,Z 758.546,A 0.000,B 0.000,C 90.000,E1 314.271} C_DIS
LIN {X 0.028,Y -684.435,Z 758.537,A 0.000,B 0.000,C 90.000,E1 312.567} C_DIS
LIN {X 0.256,Y -686.230,Z 758.531,A 0.000,B 0.000,C 90.000,E1 311.595} C_DIS
LIN {X -0.352,Y -688.273,Z 758.525,A 0.000,B 0.000,C 90.000,E1 310.458} C_DIS
LIN {X -0.401,Y -689.919,Z 758.518,A 0.000,B 0.000,C 90.000,E1 309.277} C_DIS
LIN {X 0.182,Y -691.638,Z 758.510,A 0.000,B 0.000,C 90.000,E1 307.810} C_DIS
LIN {X -0.237,Y -692.906,Z 758.504,A 0.000,B 0.000,C 90.000,E1 306.664} C_DIS
LIN {X 0.071,Y -693.571,Z 758.500,A 0.000,B 0.000,C 90.000,E1 305.931} C_DIS
LIN {X 0.107,Y -694.962,Z 758.491,A 0.000,B 0.000,C 90.000,E1 304.278} C_DIS
LIN {X -0.051,Y -696.031,Z 758.483,A 0.000,B 0.000,C 90.000,E1 302.880} C_DIS
LIN {X 0.258,Y -697.273,Z 758.474,A 0.000,B 0.000,C 90.000,E1 301.209} C_DIS
LIN {X 0.079,Y -697.886,Z 758.468,A 0.000,B 0.000,C 90.000,E1 300.285} C_DIS
LIN {X -0.005,Y -698.186,Z 758.464,A 0.000,B 0.000,C 90.000,E1 299.589} C_DIS
LIN {X -0.339,Y -698.748,Z 758.455,A 0.000,B 0.000,C 90.000,E1 297.975} C_DIS
LIN {X -0.023,Y -699.419,Z 758.446,A 0.000,B 0.000,C 90.000,E1 296.309} C_DIS
LIN {X -0.236,Y -700.012,Z 758.440,A 0.000,B 0.000,C 90.000,E1 295.155} C_DIS
LIN {X 0.304,Y -700.099,Z 758.437,A 0.000,B 0.000,C 90.000,E1 294.643} C_DIS
LIN {X -0.084,Y -699.600,Z 758.435,A 0.000,B 0.000,C 90.000,E1 294.207} C_DIS
LIN {X 0.184,Y -699.176,Z 758.433,A 0.000,B 0.000,C 90.000,E1 293.951} C_DIS
LIN {X 0.168,Y -698.265,Z 758.432,A 0.000,B 0.000,C 90.000,E1 293.718} C_DIS
LIN {X -0.077,Y -696.527,Z 758.430,A 0.000,B 0.000,C 90.000,E1 293.387} C_DIS
LIN {X 0.053,Y -695.709,Z 758.429,A 0.000,B 0.000,C 90.000,E1 293.259} C_DIS
LIN {X 0.179,Y -694.492,Z 758.429,A 0.000,B 0.000,C 90.000,E1 293.131} C_DIS
LIN {X 0.091,Y -689.823,Z 758.427,A 0.000,B 0.000,C 90.000,E1 292.823} C_DIS
LIN {X -0.392,Y -688.365,Z 758.426,A 0.000,B 0.000,C 90.000,E1 292.770} C_DIS
LIN {X 0.027,Y -686.572,Z 758.426,A 0.000,B 0.000,C 90.000,E1 292.642} C_DIS
LIN {X -0.311,Y -684.231,Z 758.425,A 0.000,B 0.000,C 90.000,E1 292.589} C_DIS
LIN {X 0.093,Y -675.785,Z 758.424,A 0.000,B 0.000,C 90.000,E1 292.333} C_DIS
LIN {X 0.290,Y -668.897,Z 758.424,A 0.000,B 0.000,C 90.000,E1 292.206} C_DIS
LIN {X 0.276,Y -653.938,Z 758.423,A 0.000,B 0.000,C 90.000,E1 292.025} C_DIS
LIN {X -0.013,Y -647.319,Z 758.422,A 0.000,B 0.000,C 90.000,E1 291.950} C_DIS
LIN {X -0.043,Y -637.835,Z 758.421,A 0.000,B 0.000,C 90.000,E1 291.770} C_DIS
LIN {X 0.005,Y -624.463,Z 758.419,A 0.000,B 0.000,C 90.000,E1 291.461} C_DIS
LIN {X -0.210,Y -607.087,Z 758.417,A 0.000,B 0.000,C 90.000,E1 291.046} C_DIS
LIN {X 0.167,Y -575.657,Z 758.412,A 0.000,B 0.000,C 90.000,E1 290.120} C_DIS
LIN {X 0.019,Y -566.717,Z 758.411,A 0.000,B 0.000,C 90.000,E1 289.885} C_DIS
LIN {X -0.074,Y -561.539,Z 758.409,A 0.000,B 0.000,C 90.000,E1 289.704} C_DIS
LIN {X -0.197,Y -558.676,Z 758.409,A 0.000,B 0.000,C 90.000,E1 289.577} C_DIS
LIN {X 0.088,Y -557.868,Z 758.408,A 0.000,B 0.000,C 90.000,E1 289.504} C_DIS
LIN {X 0.087,Y -555.833,Z 758.407,A 0.000,B 0.000,C 90.000,E1 289.268} C_DIS
LIN {X 0.171,Y -555.386,Z 758.406,A 0.000,B 0.000,C 90.000,E1 289.087} C_DIS
LIN {X 0.052,Y -555.158,Z 758.405,A 0.000,B 0.000,C 90.000,E1 288.960} C_DIS
LIN {X -0.234,Y -554.530,Z 758.397,A 0.000,B 0.000,C 90.000,E1 287.457} C_DIS
LIN {X -0.286,Y -553.877,Z 758.388,A 0.000,B 0.000,C 90.000,E1 285.788} C_DIS
LIN {X -0.235,Y -553.139,Z 758.377,A 0.000,B 0.000,C 90.000,E1 283.828} C_DIS
LIN {X 0.072,Y -552.606,Z 758.367,A 0.000,B 0.000,C 90.000,E1 282.119} C_DIS
LIN {X 0.126,Y -552.126,Z 758.360,A 0.000,B 0.000,C 90.000,E1 280.715} C_DIS
LIN {X 0.184,Y -551.492,Z 758.350,A 0.000,B 0.000,C 90.000,E1 279.029} C_DIS
LIN {X 0.183,Y -550.716,Z 758.339,A 0.000,B 0.000,C 90.000,E1 277.068} C_DIS
LIN {X -0.014,Y -550.168,Z 758.333,A 0.000,B 0.000,C 90.000,E1 275.967} C_DIS
LIN {X -0.195,Y -549.137,Z 758.324,A 0.000,B 0.000,C 90.000,E1 274.302} C_DIS
LIN {X 0.250,Y -547.828,Z 758.311,A 0.000,B 0.000,C 90.000,E1 272.007} C_DIS
LIN {X -0.002,Y -546.899,Z 758.302,A 0.000,B 0.000,C 90.000,E1 270.344} C_DIS
LIN {X -0.250,Y -545.552,Z 758.291,A 0.000,B 0.000,C 90.000,E1 268.396} C_DIS
LIN {X 0.014,Y -544.471,Z 758.282,A 0.000,B 0.000,C 90.000,E1 266.674} C_DIS
LIN {X -0.256,Y -543.268,Z 758.271,A 0.000,B 0.000,C 90.000,E1 264.723} C_DIS
LIN {X 0.002,Y -542.045,Z 758.261,A 0.000,B 0.000,C 90.000,E1 262.996} C_DIS
LIN {X 0.223,Y -541.108,Z 758.255,A 0.000,B 0.000,C 90.000,E1 261.837} C_DIS
LIN {X 0.048,Y -539.680,Z 758.245,A 0.000,B 0.000,C 90.000,E1 260.151} C_DIS
LIN {X -0.227,Y -538.541,Z 758.237,A 0.000,B 0.000,C 90.000,E1 258.757} C_DIS
LIN {X 0.101,Y -537.320,Z 758.230,A 0.000,B 0.000,C 90.000,E1 257.297} C_DIS
LIN {X -0.001,Y -536.044,Z 758.222,A 0.000,B 0.000,C 90.000,E1 255.880} C_DIS
LIN {X 0.062,Y -534.153,Z 758.212,A 0.000,B 0.000,C 90.000,E1 254.157} C_DIS
LIN {X -0.241,Y -531.886,Z 758.201,A 0.000,B 0.000,C 90.000,E1 252.181} C_DIS
LIN {X -0.324,Y -530.582,Z 758.195,A 0.000,B 0.000,C 90.000,E1 251.040} C_DIS
LIN {X -0.071,Y -528.641,Z 758.187,A 0.000,B 0.000,C 90.000,E1 249.571} C_DIS
LIN {X -0.166,Y -526.246,Z 758.177,A 0.000,B 0.000,C 90.000,E1 247.847} C_DIS
LIN {X 0.048,Y -523.150,Z 758.166,A 0.000,B 0.000,C 90.000,E1 245.793} C_DIS
LIN {X 0.093,Y -520.761,Z 758.158,A 0.000,B 0.000,C 90.000,E1 244.332} C_DIS
LIN {X 0.093,Y -518.303,Z 758.149,A 0.000,B 0.000,C 90.000,E1 242.871} C_DIS
LIN {X -0.084,Y -516.148,Z 758.143,A 0.000,B 0.000,C 90.000,E1 241.719} C_DIS
LIN {X -0.146,Y -513.339,Z 758.135,A 0.000,B 0.000,C 90.000,E1 240.255} C_DIS
LIN {X -0.152,Y -511.034,Z 758.128,A 0.000,B 0.000,C 90.000,E1 239.076} C_DIS
LIN {X 0.063,Y -508.852,Z 758.122,A 0.000,B 0.000,C 90.000,E1 237.867} C_DIS
LIN {X -0.184,Y -506.303,Z 758.115,A 0.000,B 0.000,C 90.000,E1 236.707} C_DIS
LIN {X -0.078,Y -504.378,Z 758.110,A 0.000,B 0.000,C 90.000,E1 235.801} C_DIS
LIN {X 0.188,Y -500.922,Z 758.102,A 0.000,B 0.000,C 90.000,E1 234.276} C_DIS
LIN {X 0.273,Y -497.134,Z 758.093,A 0.000,B 0.000,C 90.000,E1 232.763} C_DIS
LIN {X 0.141,Y -492.554,Z 758.083,A 0.000,B 0.000,C 90.000,E1 230.964} C_DIS
LIN {X -0.017,Y -487.556,Z 758.071,A 0.000,B 0.000,C 90.000,E1 228.852} C_DIS
LIN {X 0.210,Y -483.472,Z 758.061,A 0.000,B 0.000,C 90.000,E1 226.986} C_DIS
LIN {X -0.006,Y -479.508,Z 758.051,A 0.000,B 0.000,C 90.000,E1 225.162} C_DIS
LIN {X 0.020,Y -475.634,Z 758.041,A 0.000,B 0.000,C 90.000,E1 223.299} C_DIS
LIN {X -0.121,Y -472.246,Z 758.032,A 0.000,B 0.000,C 90.000,E1 221.757} C_DIS
LIN {X 0.291,Y -466.735,Z 758.018,A 0.000,B 0.000,C 90.000,E1 219.197} C_DIS
LIN {X -0.006,Y -463.957,Z 758.011,A 0.000,B 0.000,C 90.000,E1 217.971} C_DIS
LIN {X 0.057,Y -460.657,Z 758.002,A 0.000,B 0.000,C 90.000,E1 216.377} C_DIS
LIN {X -0.112,Y -456.796,Z 757.992,A 0.000,B 0.000,C 90.000,E1 214.485} C_DIS
LIN {X 0.004,Y -452.938,Z 757.981,A 0.000,B 0.000,C 90.000,E1 212.546} C_DIS
LIN {X 0.159,Y -449.285,Z 757.970,A 0.000,B 0.000,C 90.000,E1 210.590} C_DIS
LIN {X -0.158,Y -444.989,Z 757.957,A 0.000,B 0.000,C 90.000,E1 208.359} C_DIS
LIN {X -0.139,Y -442.587,Z 757.950,A 0.000,B 0.000,C 90.000,E1 207.052} C_DIS
LIN {X -0.094,Y -438.865,Z 757.939,A 0.000,B 0.000,C 90.000,E1 205.079} C_DIS
LIN {X 0.081,Y -435.145,Z 757.928,A 0.000,B 0.000,C 90.000,E1 203.078} C_DIS
LIN {X 0.000,Y -431.463,Z 757.917,A 0.000,B 0.000,C 90.000,E1 201.099} C_DIS
LIN {X -0.120,Y -427.025,Z 757.904,A 0.000,B 0.000,C 90.000,E1 198.779} C_DIS
LIN {X -0.073,Y -423.827,Z 757.895,A 0.000,B 0.000,C 90.000,E1 197.094} C_DIS
LIN {X -0.213,Y -420.486,Z 757.886,A 0.000,B 0.000,C 90.000,E1 195.426} C_DIS
LIN {X -0.128,Y -414.741,Z 757.869,A 0.000,B 0.000,C 90.000,E1 192.355} C_DIS
LIN {X -0.168,Y -410.654,Z 757.855,A 0.000,B 0.000,C 90.000,E1 189.962} C_DIS
LIN {X -0.033,Y -407.688,Z 757.846,A 0.000,B 0.000,C 90.000,E1 188.219} C_DIS
LIN {X -0.058,Y -403.687,Z 757.832,A 0.000,B 0.000,C 90.000,E1 185.796} C_DIS
LIN {X 0.109,Y -399.504,Z 757.817,A 0.000,B 0.000,C 90.000,E1 182.980} C_DIS
LIN {X -0.173,Y -394.143,Z 757.793,A 0.000,B 0.000,C 90.000,E1 178.797} C_DIS
LIN {X -0.053,Y -392.556,Z 757.785,A 0.000,B 0.000,C 90.000,E1 177.364} C_DIS
LIN {X 0.068,Y -389.488,Z 757.768,A 0.000,B 0.000,C 90.000,E1 174.147} C_DIS
LIN {X 0.130,Y -387.156,Z 757.748,A 0.000,B 0.000,C 90.000,E1 170.566} C_DIS
LIN {X -0.064,Y -386.359,Z 757.740,A 0.000,B 0.000,C 90.000,E1 169.162} C_DIS
LIN {X -0.022,Y -385.202,Z 757.726,A 0.000,B 0.000,C 90.000,E1 166.645} C_DIS
LIN {X 0.171,Y -383.959,Z 757.710,A 0.000,B 0.000,C 90.000,E1 163.740} C_DIS
LIN {X 0.145,Y -383.294,Z 757.698,A 0.000,B 0.000,C 90.000,E1 161.583} C_DIS
LIN {X 0.010,Y -382.643,Z 757.680,A 0.000,B 0.000,C 90.000,E1 158.358} C_DIS
LIN {X -0.079,Y -382.439,Z 757.666,A 0.000,B 0.000,C 90.000,E1 155.845} C_DIS
LIN {X -0.086,Y -383.548,Z 757.638,A 0.000,B 0.000,C 90.000,E1 150.795} C_DIS
LIN {X -0.082,Y -385.709,Z 757.622,A 0.000,B 0.000,C 90.000,E1 147.916} C_DIS
LIN {X -0.127,Y -388.739,Z 757.606,A 0.000,B 0.000,C 90.000,E1 145.055} C_DIS
LIN {X -0.186,Y -392.246,Z 757.594,A 0.000,B 0.000,C 90.000,E1 142.924} C_DIS
LIN {X 0.059,Y -394.712,Z 757.588,A 0.000,B 0.000,C 90.000,E1 141.823} C_DIS
LIN {X -0.008,Y -396.729,Z 757.584,A 0.000,B 0.000,C 90.000,E1 141.126} C_DIS
LIN {X 0.090,Y -398.578,Z 757.581,A 0.000,B 0.000,C 90.000,E1 140.598} C_DIS
LIN {X -0.013,Y -399.318,Z 757.580,A 0.000,B 0.000,C 90.000,E1 140.436} C_DIS
LIN {X -0.150,Y -401.259,Z 757.578,A 0.000,B 0.000,C 90.000,E1 140.070} C_DIS
LIN {X -0.035,Y -403.025,Z 757.576,A 0.000,B 0.000,C 90.000,E1 139.703} C_DIS
LIN {X 0.142,Y -406.058,Z 757.574,A 0.000,B 0.000,C 90.000,E1 139.218} C_DIS
LIN {X -0.026,Y -409.700,Z 757.571,A 0.000,B 0.000,C 90.000,E1 138.771} C_DIS
LIN {X -0.034,Y -416.699,Z 757.567,A 0.000,B 0.000,C 90.000,E1 138.000} C_DIS
LIN {X 0.151,Y -433.867,Z 757.557,A 0.000,B 0.000,C 90.000,E1 136.215} C_DIS
LIN {X 0.050,Y -444.077,Z 757.551,A 0.000,B 0.000,C 90.000,E1 135.202} C_DIS
LIN {X -0.002,Y -451.181,Z 757.547,A 0.000,B 0.000,C 90.000,E1 134.474} C_DIS
LIN {X 0.274,Y -458.137,Z 757.543,A 0.000,B 0.000,C 90.000,E1 133.704} C_DIS
LIN {X 0.129,Y -467.553,Z 757.537,A 0.000,B 0.000,C 90.000,E1 132.690} C_DIS
LIN {X 0.262,Y -475.533,Z 757.532,A 0.000,B 0.000,C 90.000,E1 131.757} C_DIS
LIN {X 0.294,Y -480.736,Z 757.529,A 0.000,B 0.000,C 90.000,E1 131.148} C_DIS
LIN {X 0.192,Y -489.356,Z 757.523,A 0.000,B 0.000,C 90.000,E1 130.092} C_DIS
LIN {X -0.226,Y -497.037,Z 757.517,A 0.000,B 0.000,C 90.000,E1 129.116} C_DIS
LIN {X 0.205,Y -501.301,Z 757.514,A 0.000,B 0.000,C 90.000,E1 128.463} C_DIS
LIN {X 0.067,Y -506.256,Z 757.510,A 0.000,B 0.000,C 90.000,E1 127.729} C_DIS
LIN {X -0.031,Y -510.866,Z 757.506,A 0.000,B 0.000,C 90.000,E1 126.996} C_DIS
LIN {X 0.209,Y -514.419,Z 757.502,A 0.000,B 0.000,C 90.000,E1 126.377} C_DIS
LIN {X -0.059,Y -521.076,Z 757.496,A 0.000,B 0.000,C 90.000,E1 125.231} C_DIS
LIN {X -0.108,Y -526.852,Z 757.489,A 0.000,B 0.000,C 90.000,E1 124.072} C_DIS
LIN {X -0.010,Y -528.872,Z 757.487,A 0.000,B 0.000,C 90.000,E1 123.627} C_DIS
LIN {X 0.054,Y -533.931,Z 757.480,A 0.000,B 0.000,C 90.000,E1 122.467} C_DIS
LIN {X 0.046,Y -538.071,Z 757.475,A 0.000,B 0.000,C 90.000,E1 121.465} C_DIS
LIN {X -0.240,Y -540.400,Z 757.472,A 0.000,B 0.000,C 90.000,E1 120.924} C_DIS
LIN {X -0.039,Y -543.533,Z 757.467,A 0.000,B 0.000,C 90.000,E1 120.050} C_DIS
LIN {X -0.327,Y -547.387,Z 757.461,A 0.000,B 0.000,C 90.000,E1 118.949} C_DIS
LIN {X 0.190,Y -551.077,Z 757.454,A 0.000,B 0.000,C 90.000,E1 117.769} C_DIS
LIN {X -0.277,Y -552.814,Z 757.451,A 0.000,B 0.000,C 90.000,E1 117.257} C_DIS
LIN {X 0.284,Y -555.118,Z 757.447,A 0.000,B 0.000,C 90.000,E1 116.360} C_DIS
LIN {X 0.130,Y -557.070,Z 757.442,A 0.000,B 0.000,C 90.000,E1 115.540} C_DIS
LIN {X -0.001,Y -558.737,Z 757.437,A 0.000,B 0.000,C 90.000,E1 114.719} C_DIS
LIN {X -0.115,Y -560.144,Z 757.433,A 0.000,B 0.000,C 90.000,E1 113.898} C_DIS
LIN {X -0.109,Y -562.162,Z 757.425,A 0.000,B 0.000,C 90.000,E1 112.514} C_DIS
LIN {X -0.090,Y -563.616,Z 757.419,A 0.000,B 0.000,C 90.000,E1 111.408} C_DIS
LIN {X -0.120,Y -565.708,Z 757.410,A 0.000,B 0.000,C 90.000,E1 109.758} C_DIS
LIN {X 0.092,Y -567.263,Z 757.402,A 0.000,B 0.000,C 90.000,E1 108.362} C_DIS
LIN {X 0.157,Y -568.670,Z 757.394,A 0.000,B 0.000,C 90.000,E1 106.985} C_DIS
LIN {X 0.071,Y -569.742,Z 757.388,A 0.000,B 0.000,C 90.000,E1 105.898} C_DIS
LIN {X 0.206,Y -571.400,Z 757.379,A 0.000,B 0.000,C 90.000,E1 104.245} C_DIS
LIN {X 0.215,Y -573.558,Z 757.367,A 0.000,B 0.000,C 90.000,E1 102.063} C_DIS
LIN {X 0.194,Y -575.256,Z 757.358,A 0.000,B 0.000,C 90.000,E1 100.433} C_DIS
LIN {X 0.214,Y -576.842,Z 757.349,A 0.000,B 0.000,C 90.000,E1 98.803} C_DIS
LIN {X 0.171,Y -578.215,Z 757.340,A 0.000,B 0.000,C 90.000,E1 97.182} C_DIS
LIN {X 0.086,Y -579.561,Z 757.331,A 0.000,B 0.000,C 90.000,E1 95.568} C_DIS
LIN {X -0.184,Y -580.533,Z 757.324,A 0.000,B 0.000,C 90.000,E1 94.245} C_DIS
LIN {X -0.278,Y -581.627,Z 757.315,A 0.000,B 0.000,C 90.000,E1 92.636} C_DIS
LIN {X -0.206,Y -582.749,Z 757.304,A 0.000,B 0.000,C 90.000,E1 90.745} C_DIS
LIN {X 0.105,Y -583.384,Z 757.297,A 0.000,B 0.000,C 90.000,E1 89.370} C_DIS
LIN {X 0.241,Y -583.779,Z 757.291,A 0.000,B 0.000,C 90.000,E1 88.282} C_DIS
LIN {X 0.205,Y -584.335,Z 757.282,A 0.000,B 0.000,C 90.000,E1 86.674} C_DIS
LIN {X -0.208,Y -584.573,Z 757.276,A 0.000,B 0.000,C 90.000,E1 85.641} C_DIS
LIN {X -0.227,Y -584.865,Z 757.267,A 0.000,B 0.000,C 90.000,E1 84.033} C_DIS
LIN {X 0.225,Y -584.984,Z 757.259,A 0.000,B 0.000,C 90.000,E1 82.648} C_DIS
LIN {X -0.238,Y -585.086,Z 757.250,A 0.000,B 0.000,C 90.000,E1 81.084} C_DIS
LIN {X -0.271,Y -584.933,Z 757.243,A 0.000,B 0.000,C 90.000,E1 79.746} C_DIS
LIN {X -0.069,Y -584.619,Z 757.234,A 0.000,B 0.000,C 90.000,E1 78.117} C_DIS
LIN {X -0.244,Y -584.316,Z 757.228,A 0.000,B 0.000,C 90.000,E1 77.061} C_DIS
LIN {X 0.188,Y -583.778,Z 757.219,A 0.000,B 0.000,C 90.000,E1 75.408} C_DIS
LIN {X -0.131,Y -582.916,Z 757.209,A 0.000,B 0.000,C 90.000,E1 73.559} C_DIS
LIN {X -0.136,Y -581.979,Z 757.200,A 0.000,B 0.000,C 90.000,E1 71.945} C_DIS
LIN {X -0.190,Y -581.127,Z 757.192,A 0.000,B 0.000,C 90.000,E1 70.604} C_DIS
LIN {X 0.140,Y -579.958,Z 757.183,A 0.000,B 0.000,C 90.000,E1 68.954} C_DIS
LIN {X -0.123,Y -579.006,Z 757.177,A 0.000,B 0.000,C 90.000,E1 67.901} C_DIS
LIN {X -0.159,Y -577.461,Z 757.168,A 0.000,B 0.000,C 90.000,E1 66.282} C_DIS
LIN {X -0.242,Y -575.511,Z 757.159,A 0.000,B 0.000,C 90.000,E1 64.665} C_DIS
LIN {X 0.068,Y -574.410,Z 757.155,A 0.000,B 0.000,C 90.000,E1 63.819} C_DIS
LIN {X -0.044,Y -572.759,Z 757.149,A 0.000,B 0.000,C 90.000,E1 62.743} C_DIS
LIN {X 0.077,Y -570.870,Z 757.143,A 0.000,B 0.000,C 90.000,E1 61.641} C_DIS
LIN {X -0.156,Y -569.268,Z 757.138,A 0.000,B 0.000,C 90.000,E1 60.845} C_DIS
LIN {X -0.088,Y -566.817,Z 757.132,A 0.000,B 0.000,C 90.000,E1 59.744} C_DIS
LIN {X -0.071,Y -564.788,Z 757.127,A 0.000,B 0.000,C 90.000,E1 58.918} C_DIS
LIN {X 0.211,Y -561.750,Z 757.121,A 0.000,B 0.000,C 90.000,E1 57.788} C_DIS
LIN {X 0.185,Y -559.209,Z 757.117,A 0.000,B 0.000,C 90.000,E1 56.962} C_DIS
LIN {X 0.052,Y -557.448,Z 757.114,A 0.000,B 0.000,C 90.000,E1 56.421} C_DIS
LIN {X -0.019,Y -554.552,Z 757.109,A 0.000,B 0.000,C 90.000,E1 55.595} C_DIS
LIN {X -0.122,Y -551.306,Z 757.104,A 0.000,B 0.000,C 90.000,E1 54.769} C_DIS
LIN {X -0.132,Y -548.316,Z 757.100,A 0.000,B 0.000,C 90.000,E1 54.069} C_DIS
LIN {X 0.152,Y -544.996,Z 757.096,A 0.000,B 0.000,C 90.000,E1 53.336} C_DIS
LIN {X 0.227,Y -542.182,Z 757.093,A 0.000,B 0.000,C 90.000,E1 52.763} C_DIS
LIN {X 0.125,Y -538.369,Z 757.089,A 0.000,B 0.000,C 90.000,E1 52.065} C_DIS
LIN {X -0.272,Y -535.014,Z 757.086,A 0.000,B 0.000,C 90.000,E1 51.537} C_DIS
LIN {X 0.063,Y -531.273,Z 757.083,A 0.000,B 0.000,C 90.000,E1 50.928} C_DIS
LIN {X 0.034,Y -527.165,Z 757.080,A 0.000,B 0.000,C 90.000,E1 50.356} C_DIS
LIN {X -0.029,Y -522.543,Z 757.077,A 0.000,B 0.000,C 90.000,E1 49.784} C_DIS
LIN {X -0.074,Y -517.524,Z 757.073,A 0.000,B 0.000,C 90.000,E1 49.218} C_DIS
LIN {X 0.274,Y -513.567,Z 757.071,A 0.000,B 0.000,C 90.000,E1 48.771} C_DIS
LIN {X 0.175,Y -507.784,Z 757.068,A 0.000,B 0.000,C 90.000,E1 48.243} C_DIS
LIN {X -0.092,Y -501.760,Z 757.065,A 0.000,B 0.000,C 90.000,E1 47.757} C_DIS
LIN {X -0.111,Y -497.203,Z 757.063,A 0.000,B 0.000,C 90.000,E1 47.391} C_DIS
LIN {X 0.022,Y -490.869,Z 757.061,A 0.000,B 0.000,C 90.000,E1 46.905} C_DIS
LIN {X -0.246,Y -482.820,Z 757.058,A 0.000,B 0.000,C 90.000,E1 46.377} C_DIS
LIN {X 0.133,Y -469.853,Z 757.053,A 0.000,B 0.000,C 90.000,E1 45.486} C_DIS
LIN {X -0.132,Y -452.009,Z 757.046,A 0.000,B 0.000,C 90.000,E1 44.352} C_DIS
LIN {X 0.028,Y -434.189,Z 757.040,A 0.000,B 0.000,C 90.000,E1 43.137} C_DIS
LIN {X 0.104,Y -424.810,Z 757.036,A 0.000,B 0.000,C 90.000,E1 42.447} C_DIS
LIN {X 0.112,Y -418.807,Z 757.033,A 0.000,B 0.000,C 90.000,E1 42.000} C_DIS
LIN {X -0.044,Y -413.229,Z 757.031,A 0.000,B 0.000,C 90.000,E1 41.553} C_DIS
LIN {X 0.118,Y -410.874,Z 757.030,A 0.000,B 0.000,C 90.000,E1 41.310} C_DIS
LIN {X 0.086,Y -410.864,Z 757.030,A 0.000,B 0.000,C 90.000,E1 41.310} C_DIS
LIN {X 0.010,Y -406.091,Z 757.015,A 0.000,B 0.000,C 90.000,E1 38.624} C_DIS
LIN {X -0.134,Y -403.867,Z 757.009,A 0.000,B 0.000,C 90.000,E1 37.604} C_DIS
LIN {X 0.041,Y -400.659,Z 757.000,A 0.000,B 0.000,C 90.000,E1 36.011} C_DIS
LIN {X -0.063,Y -400.440,Z 756.999,A 0.000,B 0.000,C 90.000,E1 35.851} C_DIS
LIN {X 0.057,Y -401.136,Z 756.979,A 0.000,B 0.000,C 90.000,E1 32.163} C_DIS
LIN {X -0.252,Y -402.354,Z 756.963,A 0.000,B 0.000,C 90.000,E1 29.411} C_DIS
LIN {X -0.224,Y -403.846,Z 756.948,A 0.000,B 0.000,C 90.000,E1 26.616} C_DIS
LIN {X -0.058,Y -405.913,Z 756.930,A 0.000,B 0.000,C 90.000,E1 23.462} C_DIS
LIN {X -0.135,Y -407.974,Z 756.917,A 0.000,B 0.000,C 90.000,E1 21.046} C_DIS
LIN {X 0.216,Y -409.782,Z 756.907,A 0.000,B 0.000,C 90.000,E1 19.268} C_DIS
LIN {X -0.048,Y -413.172,Z 756.892,A 0.000,B 0.000,C 90.000,E1 16.551} C_DIS
LIN {X -0.156,Y -417.131,Z 756.877,A 0.000,B 0.000,C 90.000,E1 13.828} C_DIS
LIN {X -0.106,Y -419.841,Z 756.867,A 0.000,B 0.000,C 90.000,E1 12.119} C_DIS
LIN {X -0.023,Y -423.075,Z 756.856,A 0.000,B 0.000,C 90.000,E1 10.074} C_DIS
LIN {X -0.001,Y -426.387,Z 756.845,A 0.000,B 0.000,C 90.000,E1 8.049} C_DIS
LIN {X 0.053,Y -429.711,Z 756.834,A 0.000,B 0.000,C 90.000,E1 6.030} C_DIS
LIN {X 0.020,Y -435.024,Z 756.817,A 0.000,B 0.000,C 90.000,E1 3.037} C_DIS
LIN {X -0.147,Y -439.368,Z 756.804,A 0.000,B 0.000,C 90.000,E1 0.745} C_DIS
LIN {X 0.216,Y -443.778,Z 756.792,A 0.000,B 0.000,C 90.000,E1 358.453} C_DIS
LIN {X 0.170,Y -447.970,Z 756.781,A 0.000,B 0.000,C 90.000,E1 356.502} C_DIS
LIN {X 0.168,Y -453.733,Z 756.766,A 0.000,B 0.000,C 90.000,E1 353.913} C_DIS
LIN {X 0.224,Y -457.477,Z 756.757,A 0.000,B 0.000,C 90.000,E1 352.299} C_DIS
LIN {X 0.168,Y -460.291,Z 756.750,A 0.000,B 0.000,C 90.000,E1 351.027} C_DIS
LIN {X 0.228,Y -463.010,Z 756.743,A 0.000,B 0.000,C 90.000,E1 349.746} C_DIS
LIN {X 0.133,Y -466.158,Z 756.734,A 0.000,B 0.000,C 90.000,E1 348.173} C_DIS
LIN {X -0.078,Y -468.568,Z 756.727,A 0.000,B 0.000,C 90.000,E1 346.937} C_DIS
LIN {X 0.021,Y -471.633,Z 756.719,A 0.000,B 0.000,C 90.000,E1 345.353} C_DIS
LIN {X -0.218,Y -473.217,Z 756.715,A 0.000,B 0.000,C 90.000,E1 344.755} C_DIS
LIN {X 0.011,Y -475.285,Z 756.712,A 0.000,B 0.000,C 90.000,E1 344.102} C_DIS
LIN {X -0.031,Y -476.496,Z 756.710,A 0.000,B 0.000,C 90.000,E1 343.795} C_DIS
LIN {X -0.155,Y -478.351,Z 756.708,A 0.000,B 0.000,C 90.000,E1 343.433} C_DIS
LIN {X -0.024,Y -481.706,Z 756.705,A 0.000,B 0.000,C 90.000,E1 342.906} C_DIS
LIN {X 0.190,Y -485.638,Z 756.703,A 0.000,B 0.000,C 90.000,E1 342.417} C_DIS
LIN {X 0.158,Y -490.549,Z 756.700,A 0.000,B 0.000,C 90.000,E1 341.945} C_DIS
LIN {X -0.223,Y -497.427,Z 756.697,A 0.000,B 0.000,C 90.000,E1 341.456} C_DIS
LIN {X -0.067,Y -514.822,Z 756.690,A 0.000,B 0.000,C 90.000,E1 340.242} C_DIS
LIN {X 0.116,Y -526.042,Z 756.686,A 0.000,B 0.000,C 90.000,E1 339.518} C_DIS
LIN {X 0.158,Y -537.194,Z 756.683,A 0.000,B 0.000,C 90.000,E1 338.847} C_DIS
LIN {X 0.213,Y -540.408,Z 756.682,A 0.000,B 0.000,C 90.000,E1 338.646} C_DIS
LIN {X 0.112,Y -544.720,Z 756.680,A 0.000,B 0.000,C 90.000,E1 338.358} C_DIS
LIN {X 0.121,Y -550.556,Z 756.677,A 0.000,B 0.000,C 90.000,E1 337.922} C_DIS
LIN {X -0.033,Y -554.839,Z 756.676,A 0.000,B 0.000,C 90.000,E1 337.592} C_DIS
LIN {X -0.009,Y -560.165,Z 756.673,A 0.000,B 0.000,C 90.000,E1 337.102} C_DIS
LIN {X -0.294,Y -566.520,Z 756.669,A 0.000,B 0.000,C 90.000,E1 336.485} C_DIS
LIN {X -0.045,Y -571.411,Z 756.666,A 0.000,B 0.000,C 90.000,E1 335.921} C_DIS
LIN {X -0.012,Y -578.471,Z 756.662,A 0.000,B 0.000,C 90.000,E1 335.101} C_DIS
LIN {X 0.027,Y -586.007,Z 756.656,A 0.000,B 0.000,C 90.000,E1 334.152} C_DIS
LIN {X 0.155,Y -593.081,Z 756.651,A 0.000,B 0.000,C 90.000,E1 333.204} C_DIS
LIN {X 0.111,Y -599.884,Z 756.646,A 0.000,B 0.000,C 90.000,E1 332.281} C_DIS
LIN {X -0.102,Y -605.434,Z 756.642,A 0.000,B 0.000,C 90.000,E1 331.513} C_DIS
LIN {X 0.009,Y -611.597,Z 756.637,A 0.000,B 0.000,C 90.000,E1 330.589} C_DIS
LIN {X 0.173,Y -619.099,Z 756.630,A 0.000,B 0.000,C 90.000,E1 329.410} C_DIS
LIN {X -0.086,Y -624.563,Z 756.625,A 0.000,B 0.000,C 90.000,E1 328.535} C_DIS
LIN {X -0.285,Y -629.812,Z 756.620,A 0.000,B 0.000,C 90.000,E1 327.661} C_DIS
LIN {X 0.085,Y -633.219,Z 756.617,A 0.000,B 0.000,C 90.000,E1 326.993} C_DIS
